LIN {X 0,Y 390.31,Z 233.363,A -85,B 0,C 180,E1 -11523.097,E2 -11523.097} C_VEL
LIN {X 0,Y 390.299,Z 233.363,A -85,B 0,C 180,E1 -11526.203,E2 -11526.203} C_VEL
LIN {X 0,Y 390.192,Z 233.354,A -85,B 0,C 180,E1 -11529.33,E2 -11529.33} C_VEL
LIN {X 0,Y 390.171,Z 233.375,A -85,B 0,C 180,E1 -11532.484,E2 -11532.484} C_VEL
LIN {X 0,Y 390.139,Z 233.38,A -85,B 0,C 180,E1 -11535.677,E2 -11535.677} C_VEL
LIN {X 0,Y 390.102,Z 233.369,A -85,B 0,C 180,E1 -11538.923,E2 -11538.923} C_VEL
LIN {X 0,Y 390.038,Z 233.396,A -85,B 0,C 180,E1 -11542.235,E2 -11542.235} C_VEL
LIN {X 0,Y 390.12,Z 233.376,A -85,B 0,C 180,E1 -11545.744,E2 -11545.744} C_VEL
LIN {X 0,Y 390.06,Z 233.395,A -85,B 0,C 180,E1 -11549.11,E2 -11549.11} C_VEL
LIN {X 0,Y 390.042,Z 233.39,A -85,B 0,C 180,E1 -11552.722,E2 -11552.722} C_VEL
LIN {X 0,Y 390.044,Z 233.392,A -85,B 0,C 180,E1 -11555.823,E2 -11555.823} C_VEL
LIN {X 0,Y 390.068,Z 233.387,A -85,B 0,C 180,E1 -11559.218,E2 -11559.218} C_VEL
LIN {X 0,Y 390.044,Z 233.403,A -85,B 0,C 180,E1 -11562.375,E2 -11562.375} C_VEL
LIN {X 0,Y 390.046,Z 233.395,A -85,B 0,C 180,E1 -11565.355,E2 -11565.355} C_VEL
LIN {X 0,Y 390.033,Z 233.39,A -85,B 0,C 180,E1 -11568.187,E2 -11568.187} C_VEL
LIN {X 0,Y 390.093,Z 233.385,A -85,B 0,C 180,E1 -11570.908,E2 -11570.908} C_VEL
LIN {X 0,Y 390.087,Z 233.384,A -85,B 0,C 180,E1 -11574.794,E2 -11574.794} C_VEL
LIN {X 0,Y 390.029,Z 233.399,A -85,B 0,C 180,E1 -11578.496,E2 -11578.496} C_VEL
LIN {X 0,Y 390.132,Z 233.546,A -85,B 0,C 180,E1 -11579.708,E2 -11579.708} C_VEL
LIN {X 0,Y 392.069,Z 243.393,A -85,B 0,C 180,E1 -11582.8,E2 -11582.8} C_VEL
LIN {X 0,Y 392.796,Z 249.65,A -85,B 0,C 180,E1 -11584.57,E2 -11584.57} C_VEL
LIN {X 0,Y 391.779,Z 261.902,A -85,B 0,C 180,E1 -11587.87,E2 -11587.87} C_VEL
LIN {X 0,Y 391.3,Z 267.747,A -85,B 0,C 180,E1 -11589.465,E2 -11589.465} C_VEL
LIN {X 0,Y 391.873,Z 270.886,A -85,B 0,C 180,E1 -11589.615,E2 -11589.615} C_VEL
LIN {X 0,Y 396.805,Z 298.116,A -85,B 0,C 180,E1 -11590.39,E2 -11590.39} C_VEL
LIN {X 0,Y 395.827,Z 372.67,A -85,B 0,C 180,E1 -11591.764,E2 -11591.764} C_VEL
LIN {X 0,Y 395.47,Z 383.442,A -85,B 0,C 180,E1 -11592.082,E2 -11592.082} C_VEL
LIN {X 0,Y 394.955,Z 392.542,A -85,B 0,C 180,E1 -11592.459,E2 -11592.459} C_VEL
LIN {X 0,Y 394.286,Z 402.904,A -85,B 0,C 180,E1 -11593.03,E2 -11593.03} C_VEL
LIN {X 0,Y 393.646,Z 412.039,A -85,B 0,C 180,E1 -11593.669,E2 -11593.669} C_VEL
LIN {X 0,Y 392.88,Z 421.035,A -85,B 0,C 180,E1 -11594.435,E2 -11594.435} C_VEL
LIN {X 0,Y 392.16,Z 429.764,A -85,B 0,C 180,E1 -11595.337,E2 -11595.337} C_VEL
LIN {X 0,Y 391.468,Z 437.493,A -85,B 0,C 180,E1 -11596.285,E2 -11596.285} C_VEL
LIN {X 0,Y 390.908,Z 444.382,A -85,B 0,C 180,E1 -11597.277,E2 -11597.277} C_VEL
LIN {X 0,Y 390.29,Z 450.582,A -85,B 0,C 180,E1 -11598.312,E2 -11598.312} C_VEL
LIN {X 0,Y 389.786,Z 457.122,A -85,B 0,C 180,E1 -11599.613,E2 -11599.613} C_VEL
LIN {X 0,Y 389.386,Z 461.622,A -85,B 0,C 180,E1 -11600.651,E2 -11600.651} C_VEL
LIN {X 0,Y 389.018,Z 467.114,A -85,B 0,C 180,E1 -11602.213,E2 -11602.213} C_VEL
LIN {X 0,Y 388.796,Z 471.439,A -85,B 0,C 180,E1 -11603.774,E2 -11603.774} C_VEL
LIN {X 0,Y 388.74,Z 473.806,A -85,B 0,C 180,E1 -11604.814,E2 -11604.814} C_VEL
LIN {X 0,Y 388.7,Z 475.604,A -85,B 0,C 180,E1 -11605.853,E2 -11605.853} C_VEL
LIN {X 0,Y 388.661,Z 478.048,A -85,B 0,C 180,E1 -11607.927,E2 -11607.927} C_VEL
LIN {X 0,Y 388.704,Z 478.637,A -85,B 0,C 180,E1 -11608.964,E2 -11608.964} C_VEL
LIN {X 0,Y 388.704,Z 478.637,A -85,B 0,C 180,E1 -11611.036,E2 -11611.036} C_VEL
LIN {X 0,Y 388.661,Z 478.048,A -85,B 0,C 180,E1 -11612.073,E2 -11612.073} C_VEL
LIN {X 0,Y 388.7,Z 475.604,A -85,B 0,C 180,E1 -11614.147,E2 -11614.147} C_VEL
LIN {X 0,Y 388.727,Z 472.551,A -85,B 0,C 180,E1 -11615.751,E2 -11615.751} C_VEL
LIN {X 0,Y 388.933,Z 468.668,A -85,B 0,C 180,E1 -11617.267,E2 -11617.267} C_VEL
LIN {X 0,Y 389.252,Z 463.539,A -85,B 0,C 180,E1 -11618.828,E2 -11618.828} C_VEL
LIN {X 0,Y 389.661,Z 458.277,A -85,B 0,C 180,E1 -11620.128,E2 -11620.128} C_VEL
LIN {X 0,Y 390.15,Z 451.958,A -85,B 0,C 180,E1 -11621.429,E2 -11621.429} C_VEL
LIN {X 0,Y 390.729,Z 446.008,A -85,B 0,C 180,E1 -11622.465,E2 -11622.465} C_VEL
LIN {X 0,Y 391.321,Z 439.079,A -85,B 0,C 180,E1 -11623.502,E2 -11623.502} C_VEL
LIN {X 0,Y 392.026,Z 430.898,A -85,B 0,C 180,E1 -11624.536,E2 -11624.536} C_VEL
LIN {X 0,Y 392.747,Z 422.386,A -85,B 0,C 180,E1 -11625.437,E2 -11625.437} C_VEL
LIN {X 0,Y 393.498,Z 413.67,A -85,B 0,C 180,E1 -11626.204,E2 -11626.204} C_VEL
LIN {X 0,Y 394.227,Z 403.912,A -85,B 0,C 180,E1 -11626.906,E2 -11626.906} C_VEL
LIN {X 0,Y 394.878,Z 393.83,A -85,B 0,C 180,E1 -11627.478,E2 -11627.478} C_VEL
LIN {X 0,Y 395.404,Z 384.315,A -85,B 0,C 180,E1 -11627.888,E2 -11627.888} C_VEL
LIN {X 0,Y 395.822,Z 374.003,A -85,B 0,C 180,E1 -11628.203,E2 -11628.203} C_VEL
LIN {X 0,Y 396.82,Z 301.34,A -85,B 0,C 180,E1 -11629.549,E2 -11629.549} C_VEL
LIN {X 0,Y 396.586,Z 296.789,A -85,B 0,C 180,E1 -11629.647,E2 -11629.647} C_VEL
LIN {X 0,Y 391.485,Z 269.134,A -85,B 0,C 180,E1 -11630.439,E2 -11630.439} C_VEL
LIN {X 0,Y 391.317,Z 267.542,A -85,B 0,C 180,E1 -11630.569,E2 -11630.569} C_VEL
LIN {X 0,Y 392.512,Z 253.975,A -85,B 0,C 180,E1 -11634.319,E2 -11634.319} C_VEL
LIN {X 0,Y 392.875,Z 249.939,A -85,B 0,C 180,E1 -11635.425,E2 -11635.425} C_VEL
LIN {X 0,Y 392.151,Z 243.762,A -85,B 0,C 180,E1 -11637.194,E2 -11637.194} C_VEL
LIN {X 0,Y 390.184,Z 233.887,A -85,B 0,C 180,E1 -11640.165,E2 -11640.165} C_VEL
LIN {X 0,Y 390.088,Z 233.399,A -85,B 0,C 180,E1 -11640.445,E2 -11640.445} C_VEL
LIN {X 0,Y 390.071,Z 233.398,A -85,B 0,C 180,E1 -11644.024,E2 -11644.024} C_VEL
LIN {X 0,Y 390.046,Z 233.4,A -85,B 0,C 180,E1 -11647.55,E2 -11647.55} C_VEL
LIN {X 0,Y 390.058,Z 233.377,A -85,B 0,C 180,E1 -11650.821,E2 -11650.821} C_VEL
LIN {X 0,Y 390.056,Z 233.398,A -85,B 0,C 180,E1 -11653.886,E2 -11653.886} C_VEL
LIN {X 0,Y 390.059,Z 233.394,A -85,B 0,C 180,E1 -11656.789,E2 -11656.789} C_VEL
LIN {X 0,Y 390.057,Z 233.39,A -85,B 0,C 180,E1 -11659.56,E2 -11659.56} C_VEL
LIN {X 0,Y 390.043,Z 233.397,A -85,B 0,C 180,E1 -11662.449,E2 -11662.449} C_VEL
LIN {X 0,Y 390.062,Z 233.383,A -85,B 0,C 180,E1 -11666.044,E2 -11666.044} C_VEL
LIN {X 0,Y 390.047,Z 233.397,A -85,B 0,C 180,E1 -11669.869,E2 -11669.869} C_VEL
LIN {X 0,Y 390.114,Z 233.372,A -85,B 0,C 180,E1 -11673.231,E2 -11673.231} C_VEL
LIN {X 0,Y 390.077,Z 233.392,A -85,B 0,C 180,E1 -11676.76,E2 -11676.76} C_VEL
LIN {X 0,Y 390.103,Z 233.375,A -85,B 0,C 180,E1 -11679.982,E2 -11679.982} C_VEL
LIN {X 0,Y 390.138,Z 233.375,A -85,B 0,C 180,E1 -11683.248,E2 -11683.248} C_VEL
LIN {X 0,Y 390.195,Z 233.378,A -85,B 0,C 180,E1 -11686.561,E2 -11686.561} C_VEL
LIN {X 0,Y 390.167,Z 233.358,A -85,B 0,C 180,E1 -11689.622,E2 -11689.622} C_VEL
LIN {X 0,Y 390.266,Z 233.36,A -85,B 0,C 180,E1 -11692.758,E2 -11692.758} C_VEL
LIN {X 0,Y 390.218,Z 233.379,A -85,B 0,C 180,E1 -11694.833,E2 -11694.833} C_VEL
LIN {X 0,Y 390.418,Z 233.343,A -85,B 0,C 180,E1 -11697.936,E2 -11697.936} C_VEL
LIN {X 0,Y 390.547,Z 233.31,A -85,B 0,C 180,E1 -11699.999,E2 -11699.999} C_VEL
LIN {X 0,Y 390.313,Z 233.362,A -85,B 0,C 180,E1 -11703.096,E2 -11703.096} C_VEL
LIN {X 0,Y 390.3,Z 233.362,A -85,B 0,C 180,E1 -11706.572,E2 -11706.572} C_VEL
LIN {X 0,Y 390.204,Z 233.353,A -85,B 0,C 180,E1 -11709.328,E2 -11709.328} C_VEL
LIN {X 0,Y 390.193,Z 233.377,A -85,B 0,C 180,E1 -11713.438,E2 -11713.438} C_VEL
LIN {X 0,Y 390.147,Z 233.374,A -85,B 0,C 180,E1 -11717.307,E2 -11717.307} C_VEL
LIN {X 0,Y 390.085,Z 233.379,A -85,B 0,C 180,E1 -11720.47,E2 -11720.47} C_VEL
LIN {X 0,Y 390.074,Z 233.393,A -85,B 0,C 180,E1 -11724.48,E2 -11724.48} C_VEL
LIN {X 0,Y 390.114,Z 233.371,A -85,B 0,C 180,E1 -11727.929,E2 -11727.929} C_VEL
LIN {X 0,Y 390.021,Z 233.401,A -85,B 0,C 180,E1 -11731.504,E2 -11731.504} C_VEL
LIN {X 0,Y 390.082,Z 233.382,A -85,B 0,C 180,E1 -11735.206,E2 -11735.206} C_VEL
LIN {X 0,Y 390.089,Z 233.39,A -85,B 0,C 180,E1 -11739.092,E2 -11739.092} C_VEL
LIN {X 0,Y 390.117,Z 233.39,A -85,B 0,C 180,E1 -11742.386,E2 -11742.386} C_VEL
LIN {X 0,Y 390.059,Z 233.389,A -85,B 0,C 180,E1 -11745.357,E2 -11745.357} C_VEL
LIN {X 0,Y 390.073,Z 233.371,A -85,B 0,C 180,E1 -11749.175,E2 -11749.175} C_VEL
LIN {X 0,Y 390.043,Z 233.398,A -85,B 0,C 180,E1 -11752.448,E2 -11752.448} C_VEL
LIN {X 0,Y 390.064,Z 233.377,A -85,B 0,C 180,E1 -11756.045,E2 -11756.045} C_VEL
LIN {X 0,Y 390.043,Z 233.386,A -85,B 0,C 180,E1 -11759.869,E2 -11759.869} C_VEL
LIN {X 0,Y 390.11,Z 233.394,A -85,B 0,C 180,E1 -11763.232,E2 -11763.232} C_VEL
LIN {X 0,Y 390.103,Z 233.393,A -85,B 0,C 180,E1 -11766.75,E2 -11766.75} C_VEL
LIN {X 0,Y 390.1,Z 233.395,A -85,B 0,C 180,E1 -11769.983,E2 -11769.983} C_VEL
LIN {X 0,Y 390.134,Z 233.391,A -85,B 0,C 180,E1 -11773.248,E2 -11773.248} C_VEL
LIN {X 0,Y 390.191,Z 233.383,A -85,B 0,C 180,E1 -11776.561,E2 -11776.561} C_VEL
LIN {X 0,Y 390.202,Z 233.382,A -85,B 0,C 180,E1 -11780.671,E2 -11780.671} C_VEL
LIN {X 0,Y 390.404,Z 233.767,A -85,B 0,C 180,E1 -11781.927,E2 -11781.927} C_VEL
LIN {X 0,Y 391.193,Z 235.98,A -85,B 0,C 180,E1 -11782.905,E2 -11782.905} C_VEL
LIN {X 0,Y 392.56,Z 237.719,A -85,B 0,C 180,E1 -11783.962,E2 -11783.962} C_VEL
LIN {X 0,Y 394.309,Z 239.002,A -85,B 0,C 180,E1 -11785.656,E2 -11785.656} C_VEL
LIN {X 0,Y 395.582,Z 239.492,A -85,B 0,C 180,E1 -11787.454,E2 -11787.454} C_VEL
LIN {X 0,Y 396.128,Z 239.931,A -85,B 0,C 180,E1 -11788.983,E2 -11788.983} C_VEL
LIN {X 0,Y 396.323,Z 239.849,A -85,B 0,C 180,E1 -11790,E2 -11790} C_VEL
LIN {X 0,Y 396.07,Z 239.804,A -85,B 0,C 180,E1 -11791.525,E2 -11791.525} C_VEL
LIN {X 0,Y 395.354,Z 239.371,A -85,B 0,C 180,E1 -11793.057,E2 -11793.057} C_VEL
LIN {X 0,Y 393.693,Z 238.657,A -85,B 0,C 180,E1 -11794.993,E2 -11794.993} C_VEL
LIN {X 0,Y 391.898,Z 237.018,A -85,B 0,C 180,E1 -11796.565,E2 -11796.565} C_VEL
LIN {X 0,Y 390.579,Z 234.501,A -85,B 0,C 180,E1 -11797.684,E2 -11797.684} C_VEL
LIN {X 0,Y 390.341,Z 233.593,A -85,B 0,C 180,E1 -11798.282,E2 -11798.282} C_VEL
LIN {X 0,Y 390.145,Z 233.389,A -85,B 0,C 180,E1 -11801.429,E2 -11801.429} C_VEL
LIN {X 0,Y 390.141,Z 233.39,A -85,B 0,C 180,E1 -11804.607,E2 -11804.607} C_VEL
LIN {X 0,Y 390.124,Z 233.392,A -85,B 0,C 180,E1 -11807.833,E2 -11807.833} C_VEL
LIN {X 0,Y 390.052,Z 233.401,A -85,B 0,C 180,E1 -11811.122,E2 -11811.122} C_VEL
LIN {X 0,Y 390.076,Z 233.398,A -85,B 0,C 180,E1 -11814.481,E2 -11814.481} C_VEL
LIN {X 0,Y 390.113,Z 233.387,A -85,B 0,C 180,E1 -11817.93,E2 -11817.93} C_VEL
LIN {X 0,Y 390.008,Z 233.394,A -85,B 0,C 180,E1 -11820.807,E2 -11820.807} C_VEL
LIN {X 0,Y 389.335,Z 233.489,A -85,B 0,C 180,E1 -11821.669,E2 -11821.669} C_VEL
LIN {X 0,Y 386.487,Z 233.835,A -85,B 0,C 180,E1 -11823.071,E2 -11823.071} C_VEL
LIN {X 0,Y 384.089,Z 234.122,A -85,B 0,C 180,E1 -11824.204,E2 -11824.204} C_VEL
LIN {X 0,Y 383.072,Z 234.245,A -85,B 0,C 180,E1 -11825.08,E2 -11825.08} C_VEL
LIN {X 0,Y 382.995,Z 234.255,A -85,B 0,C 180,E1 -11825.376,E2 -11825.376} C_VEL
LIN {X 0,Y 383.005,Z 234.275,A -85,B 0,C 180,E1 -11828.6,E2 -11828.6} C_VEL
LIN {X 0,Y 382.999,Z 234.243,A -85,B 0,C 180,E1 -11831.345,E2 -11831.345} C_VEL
LIN {X 0,Y 383.004,Z 234.261,A -85,B 0,C 180,E1 -11834.306,E2 -11834.306} C_VEL
LIN {X 0,Y 383.071,Z 234.266,A -85,B 0,C 180,E1 -11837.25,E2 -11837.25} C_VEL
LIN {X 0,Y 383.018,Z 234.27,A -85,B 0,C 180,E1 -11840.413,E2 -11840.413} C_VEL
LIN {X 0,Y 383.023,Z 234.266,A -85,B 0,C 180,E1 -11844.045,E2 -11844.045} C_VEL
LIN {X 0,Y 382.984,Z 234.275,A -85,B 0,C 180,E1 -11847.578,E2 -11847.578} C_VEL
LIN {X 0,Y 382.989,Z 234.273,A -85,B 0,C 180,E1 -11850.301,E2 -11850.301} C_VEL
LIN {X 0,Y 383.077,Z 234.256,A -85,B 0,C 180,E1 -11854.021,E2 -11854.021} C_VEL
LIN {X 0,Y 382.989,Z 234.279,A -85,B 0,C 180,E1 -11857.335,E2 -11857.335} C_VEL
LIN {X 0,Y 383.058,Z 234.245,A -85,B 0,C 180,E1 -11860.717,E2 -11860.717} C_VEL
LIN {X 0,Y 383.079,Z 234.265,A -85,B 0,C 180,E1 -11864.027,E2 -11864.027} C_VEL
LIN {X 0,Y 383.135,Z 234.255,A -85,B 0,C 180,E1 -11867.284,E2 -11867.284} C_VEL
LIN {X 0,Y 383.15,Z 234.231,A -85,B 0,C 180,E1 -11870.498,E2 -11870.498} C_VEL
LIN {X 0,Y 383.279,Z 234.242,A -85,B 0,C 180,E1 -11873.684,E2 -11873.684} C_VEL
LIN {X 0,Y 383.386,Z 234.213,A -85,B 0,C 180,E1 -11877.899,E2 -11877.899} C_VEL
LIN {X 0,Y 383.517,Z 234.184,A -85,B 0,C 180,E1 -11880.001,E2 -11880.001} C_VEL
LIN {X 0,Y 383.246,Z 234.243,A -85,B 0,C 180,E1 -11883.154,E2 -11883.154} C_VEL
LIN {X 0,Y 383.255,Z 234.24,A -85,B 0,C 180,E1 -11886.317,E2 -11886.317} C_VEL
LIN {X 0,Y 383.143,Z 234.231,A -85,B 0,C 180,E1 -11889.503,E2 -11889.503} C_VEL
LIN {X 0,Y 383.136,Z 234.253,A -85,B 0,C 180,E1 -11892.717,E2 -11892.717} C_VEL
LIN {X 0,Y 383.081,Z 234.259,A -85,B 0,C 180,E1 -11895.974,E2 -11895.974} C_VEL
LIN {X 0,Y 383.058,Z 234.248,A -85,B 0,C 180,E1 -11899.284,E2 -11899.284} C_VEL
LIN {X 0,Y 382.996,Z 234.277,A -85,B 0,C 180,E1 -11902.666,E2 -11902.666} C_VEL
LIN {X 0,Y 383.08,Z 234.251,A -85,B 0,C 180,E1 -11906.124,E2 -11906.124} C_VEL
LIN {X 0,Y 382.993,Z 234.274,A -85,B 0,C 180,E1 -11909.7,E2 -11909.7} C_VEL
LIN {X 0,Y 382.999,Z 234.262,A -85,B 0,C 180,E1 -11913.402,E2 -11913.402} C_VEL
LIN {X 0,Y 383.024,Z 234.269,A -85,B 0,C 180,E1 -11916.163,E2 -11916.163} C_VEL
LIN {X 0,Y 383.009,Z 234.266,A -85,B 0,C 180,E1 -11919.959,E2 -11919.959} C_VEL
LIN {X 0,Y 383.007,Z 234.275,A -85,B 0,C 180,E1 -11922.779,E2 -11922.779} C_VEL
LIN {X 0,Y 382.999,Z 234.275,A -85,B 0,C 180,E1 -11925.79,E2 -11925.79} C_VEL
LIN {X 0,Y 382.99,Z 234.26,A -85,B 0,C 180,E1 -11928.796,E2 -11928.796} C_VEL
LIN {X 0,Y 383.002,Z 234.279,A -85,B 0,C 180,E1 -11932.097,E2 -11932.097} C_VEL
LIN {X 0,Y 383.02,Z 234.269,A -85,B 0,C 180,E1 -11935.332,E2 -11935.332} C_VEL
LIN {X 0,Y 383.049,Z 234.292,A -85,B 0,C 180,E1 -11939.309,E2 -11939.309} C_VEL
LIN {X 0,Y 384.788,Z 243.209,A -85,B 0,C 180,E1 -11942.242,E2 -11942.242} C_VEL
LIN {X 0,Y 385.782,Z 249.475,A -85,B 0,C 180,E1 -11944.073,E2 -11944.073} C_VEL
LIN {X 0,Y 385.378,Z 256.646,A -85,B 0,C 180,E1 -11946.036,E2 -11946.036} C_VEL
LIN {X 0,Y 384.406,Z 267.552,A -85,B 0,C 180,E1 -11949.078,E2 -11949.078} C_VEL
LIN {X 0,Y 384.82,Z 270.202,A -85,B 0,C 180,E1 -11949.215,E2 -11949.215} C_VEL
LIN {X 0,Y 390.06,Z 298.316,A -85,B 0,C 180,E1 -11950.044,E2 -11950.044} C_VEL
LIN {X 0,Y 389.103,Z 372.478,A -85,B 0,C 180,E1 -11951.437,E2 -11951.437} C_VEL
LIN {X 0,Y 388.708,Z 383.249,A -85,B 0,C 180,E1 -11951.759,E2 -11951.759} C_VEL
LIN {X 0,Y 388.182,Z 392.349,A -85,B 0,C 180,E1 -11952.143,E2 -11952.143} C_VEL
LIN {X 0,Y 387.492,Z 402.711,A -85,B 0,C 180,E1 -11952.723,E2 -11952.723} C_VEL
LIN {X 0,Y 386.841,Z 411.846,A -85,B 0,C 180,E1 -11953.373,E2 -11953.373} C_VEL
LIN {X 0,Y 386.018,Z 420.841,A -85,B 0,C 180,E1 -11954.151,E2 -11954.151} C_VEL
LIN {X 0,Y 385.273,Z 429.571,A -85,B 0,C 180,E1 -11955.069,E2 -11955.069} C_VEL
LIN {X 0,Y 384.536,Z 437.481,A -85,B 0,C 180,E1 -11956.058,E2 -11956.058} C_VEL
LIN {X 0,Y 383.792,Z 445.815,A -85,B 0,C 180,E1 -11957.306,E2 -11957.306} C_VEL
LIN {X 0,Y 383.166,Z 451.764,A -85,B 0,C 180,E1 -11958.36,E2 -11958.36} C_VEL
LIN {X 0,Y 382.657,Z 458.083,A -85,B 0,C 180,E1 -11959.684,E2 -11959.684} C_VEL
LIN {X 0,Y 382.209,Z 463.345,A -85,B 0,C 180,E1 -11961.008,E2 -11961.008} C_VEL
LIN {X 0,Y 381.861,Z 468.474,A -85,B 0,C 180,E1 -11962.598,E2 -11962.598} C_VEL
LIN {X 0,Y 381.688,Z 471.762,A -85,B 0,C 180,E1 -11963.883,E2 -11963.883} C_VEL
LIN {X 0,Y 381.641,Z 473.612,A -85,B 0,C 180,E1 -11964.717,E2 -11964.717} C_VEL
LIN {X 0,Y 381.625,Z 475.411,A -85,B 0,C 180,E1 -11965.776,E2 -11965.776} C_VEL
LIN {X 0,Y 381.56,Z 477.855,A -85,B 0,C 180,E1 -11967.889,E2 -11967.889} C_VEL
LIN {X 0,Y 381.603,Z 478.444,A -85,B 0,C 180,E1 -11968.945,E2 -11968.945} C_VEL
LIN {X 0,Y 381.603,Z 478.444,A -85,B 0,C 180,E1 -11971.055,E2 -11971.055} C_VEL
LIN {X 0,Y 381.56,Z 477.855,A -85,B 0,C 180,E1 -11972.111,E2 -11972.111} C_VEL
LIN {X 0,Y 381.625,Z 475.411,A -85,B 0,C 180,E1 -11974.224,E2 -11974.224} C_VEL
LIN {X 0,Y 381.641,Z 473.612,A -85,B 0,C 180,E1 -11975.283,E2 -11975.283} C_VEL
LIN {X 0,Y 381.781,Z 470.005,A -85,B 0,C 180,E1 -11976.872,E2 -11976.872} C_VEL
LIN {X 0,Y 382.058,Z 465.26,A -85,B 0,C 180,E1 -11978.462,E2 -11978.462} C_VEL
LIN {X 0,Y 382.532,Z 459.238,A -85,B 0,C 180,E1 -11980.052,E2 -11980.052} C_VEL
LIN {X 0,Y 383.05,Z 453.141,A -85,B 0,C 180,E1 -11981.375,E2 -11981.375} C_VEL
LIN {X 0,Y 383.611,Z 447.441,A -85,B 0,C 180,E1 -11982.431,E2 -11982.431} C_VEL
LIN {X 0,Y 384.39,Z 438.886,A -85,B 0,C 180,E1 -11983.75,E2 -11983.75} C_VEL
LIN {X 0,Y 385.145,Z 430.705,A -85,B 0,C 180,E1 -11984.801,E2 -11984.801} C_VEL
LIN {X 0,Y 385.907,Z 422.193,A -85,B 0,C 180,E1 -11985.718,E2 -11985.718} C_VEL
LIN {X 0,Y 386.667,Z 413.477,A -85,B 0,C 180,E1 -11986.499,E2 -11986.499} C_VEL
LIN {X 0,Y 387.429,Z 403.719,A -85,B 0,C 180,E1 -11987.212,E2 -11987.212} C_VEL
LIN {X 0,Y 388.121,Z 393.637,A -85,B 0,C 180,E1 -11987.792,E2 -11987.792} C_VEL
LIN {X 0,Y 388.668,Z 384.123,A -85,B 0,C 180,E1 -11988.209,E2 -11988.209} C_VEL
LIN {X 0,Y 389.092,Z 373.81,A -85,B 0,C 180,E1 -11988.529,E2 -11988.529} C_VEL
LIN {X 0,Y 390.142,Z 301.313,A -85,B 0,C 180,E1 -11989.895,E2 -11989.895} C_VEL
LIN {X 0,Y 389.76,Z 296.708,A -85,B 0,C 180,E1 -11990.003,E2 -11990.003} C_VEL
LIN {X 0,Y 384.568,Z 268.933,A -85,B 0,C 180,E1 -11990.824,E2 -11990.824} C_VEL
LIN {X 0,Y 384.385,Z 267.342,A -85,B 0,C 180,E1 -11990.958,E2 -11990.958} C_VEL
LIN {X 0,Y 385.663,Z 253.791,A -85,B 0,C 180,E1 -11994.78,E2 -11994.78} C_VEL
LIN {X 0,Y 385.873,Z 249.767,A -85,B 0,C 180,E1 -11995.92,E2 -11995.92} C_VEL
LIN {X 0,Y 384.556,Z 241.517,A -85,B 0,C 180,E1 -11998.37,E2 -11998.37} C_VEL
LIN {X 0,Y 383.049,Z 234.295,A -85,B 0,C 180,E1 -12000.692,E2 -12000.692} C_VEL
LIN {X 0,Y 383.02,Z 234.27,A -85,B 0,C 180,E1 -12004.668,E2 -12004.668} C_VEL
LIN {X 0,Y 383.002,Z 234.279,A -85,B 0,C 180,E1 -12007.903,E2 -12007.903} C_VEL
LIN {X 0,Y 382.985,Z 234.261,A -85,B 0,C 180,E1 -12011.347,E2 -12011.347} C_VEL
LIN {X 0,Y 382.997,Z 234.274,A -85,B 0,C 180,E1 -12014.303,E2 -12014.303} C_VEL
LIN {X 0,Y 383.012,Z 234.274,A -85,B 0,C 180,E1 -12017.24,E2 -12017.24} C_VEL
LIN {X 0,Y 383.015,Z 234.266,A -85,B 0,C 180,E1 -12020.413,E2 -12020.413} C_VEL
LIN {X 0,Y 383.016,Z 234.269,A -85,B 0,C 180,E1 -12024.043,E2 -12024.043} C_VEL
LIN {X 0,Y 382.986,Z 234.273,A -85,B 0,C 180,E1 -12027.578,E2 -12027.578} C_VEL
LIN {X 0,Y 382.993,Z 234.274,A -85,B 0,C 180,E1 -12030.3,E2 -12030.3} C_VEL
LIN {X 0,Y 383.081,Z 234.253,A -85,B 0,C 180,E1 -12034.02,E2 -12034.02} C_VEL
LIN {X 0,Y 382.996,Z 234.277,A -85,B 0,C 180,E1 -12037.334,E2 -12037.334} C_VEL
LIN {X 0,Y 383.058,Z 234.248,A -85,B 0,C 180,E1 -12040.716,E2 -12040.716} C_VEL
LIN {X 0,Y 383.081,Z 234.259,A -85,B 0,C 180,E1 -12044.026,E2 -12044.026} C_VEL
LIN {X 0,Y 383.136,Z 234.253,A -85,B 0,C 180,E1 -12047.283,E2 -12047.283} C_VEL
LIN {X 0,Y 383.143,Z 234.231,A -85,B 0,C 180,E1 -12050.497,E2 -12050.497} C_VEL
LIN {X 0,Y 383.255,Z 234.24,A -85,B 0,C 180,E1 -12053.683,E2 -12053.683} C_VEL
LIN {X 0,Y 383.385,Z 234.218,A -85,B 0,C 180,E1 -12057.898,E2 -12057.898} C_VEL
LIN {X 0,Y 383.517,Z 234.184,A -85,B 0,C 180,E1 -12059.999,E2 -12059.999} C_VEL
LIN {X 0,Y 383.249,Z 234.243,A -85,B 0,C 180,E1 -12063.153,E2 -12063.153} C_VEL
LIN {X 0,Y 383.261,Z 234.24,A -85,B 0,C 180,E1 -12066.563,E2 -12066.563} C_VEL
LIN {X 0,Y 383.15,Z 234.231,A -85,B 0,C 180,E1 -12069.502,E2 -12069.502} C_VEL
LIN {X 0,Y 383.124,Z 234.257,A -85,B 0,C 180,E1 -12073.536,E2 -12073.536} C_VEL
LIN {X 0,Y 383.093,Z 234.253,A -85,B 0,C 180,E1 -12077.454,E2 -12077.454} C_VEL
LIN {X 0,Y 383.026,Z 234.26,A -85,B 0,C 180,E1 -12080.646,E2 -12080.646} C_VEL
LIN {X 0,Y 383.02,Z 234.274,A -85,B 0,C 180,E1 -12083.807,E2 -12083.807} C_VEL
LIN {X 0,Y 383.077,Z 234.254,A -85,B 0,C 180,E1 -12086.123,E2 -12086.123} C_VEL
LIN {X 0,Y 382.989,Z 234.273,A -85,B 0,C 180,E1 -12089.699,E2 -12089.699} C_VEL
LIN {X 0,Y 383,Z 234.27,A -85,B 0,C 180,E1 -12093.4,E2 -12093.4} C_VEL
LIN {X 0,Y 383.03,Z 234.268,A -85,B 0,C 180,E1 -12096.164,E2 -12096.164} C_VEL
LIN {X 0,Y 383.014,Z 234.266,A -85,B 0,C 180,E1 -12099.957,E2 -12099.957} C_VEL
LIN {X 0,Y 383.062,Z 234.267,A -85,B 0,C 180,E1 -12102.788,E2 -12102.788} C_VEL
LIN {X 0,Y 383.004,Z 234.259,A -85,B 0,C 180,E1 -12105.79,E2 -12105.79} C_VEL
LIN {X 0,Y 383.004,Z 234.244,A -85,B 0,C 180,E1 -12108.792,E2 -12108.792} C_VEL
LIN {X 0,Y 382.999,Z 234.278,A -85,B 0,C 180,E1 -12112.095,E2 -12112.095} C_VEL
LIN {X 0,Y 383.014,Z 234.251,A -85,B 0,C 180,E1 -12115.332,E2 -12115.332} C_VEL
LIN {X 0,Y 382.979,Z 234.278,A -85,B 0,C 180,E1 -12119.081,E2 -12119.081} C_VEL
LIN {X 0,Y 383.053,Z 234.27,A -85,B 0,C 180,E1 -12122.698,E2 -12122.698} C_VEL
LIN {X 0,Y 383.03,Z 234.274,A -85,B 0,C 180,E1 -12126.193,E2 -12126.193} C_VEL
LIN {X 0,Y 383.051,Z 234.273,A -85,B 0,C 180,E1 -12129.598,E2 -12129.598} C_VEL
LIN {X 0,Y 383.101,Z 234.267,A -85,B 0,C 180,E1 -12132.931,E2 -12132.931} C_VEL
LIN {X 0,Y 383.121,Z 234.263,A -85,B 0,C 180,E1 -12136.464,E2 -12136.464} C_VEL
LIN {X 0,Y 383.154,Z 234.531,A -85,B 0,C 180,E1 -12138.527,E2 -12138.527} C_VEL
LIN {X 0,Y 383.436,Z 235.716,A -85,B 0,C 180,E1 -12138.971,E2 -12138.971} C_VEL
LIN {X 0,Y 384.578,Z 237.759,A -85,B 0,C 180,E1 -12139.603,E2 -12139.603} C_VEL
LIN {X 0,Y 386.856,Z 239.64,A -85,B 0,C 180,E1 -12140.722,E2 -12140.722} C_VEL
LIN {X 0,Y 388.921,Z 240.829,A -85,B 0,C 180,E1 -12141.896,E2 -12141.896} C_VEL
LIN {X 0,Y 390.34,Z 243.395,A -85,B 0,C 180,E1 -12142.955,E2 -12142.955} C_VEL
LIN {X 0,Y 391.933,Z 245.07,A -85,B 0,C 180,E1 -12144.211,E2 -12144.211} C_VEL
LIN {X 0,Y 393.437,Z 246.033,A -85,B 0,C 180,E1 -12145.646,E2 -12145.646} C_VEL
LIN {X 0,Y 394.719,Z 246.512,A -85,B 0,C 180,E1 -12147.449,E2 -12147.449} C_VEL
LIN {X 0,Y 395.266,Z 246.977,A -85,B 0,C 180,E1 -12148.981,E2 -12148.981} C_VEL
LIN {X 0,Y 395.458,Z 246.896,A -85,B 0,C 180,E1 -12150,E2 -12150} C_VEL
LIN {X 0,Y 395.202,Z 246.853,A -85,B 0,C 180,E1 -12151.529,E2 -12151.529} C_VEL
LIN {X 0,Y 394.244,Z 246.355,A -85,B 0,C 180,E1 -12153.368,E2 -12153.368} C_VEL
LIN {X 0,Y 392.65,Z 245.62,A -85,B 0,C 180,E1 -12155.135,E2 -12155.135} C_VEL
LIN {X 0,Y 390.787,Z 243.978,A -85,B 0,C 180,E1 -12156.713,E2 -12156.713} C_VEL
LIN {X 0,Y 389.246,Z 241.409,A -85,B 0,C 180,E1 -12157.901,E2 -12157.901} C_VEL
LIN {X 0,Y 388.306,Z 240.316,A -85,B 0,C 180,E1 -12158.456,E2 -12158.456} C_VEL
LIN {X 0,Y 385.837,Z 239.007,A -85,B 0,C 180,E1 -12159.766,E2 -12159.766} C_VEL
LIN {X 0,Y 383.934,Z 236.786,A -85,B 0,C 180,E1 -12160.748,E2 -12160.748} C_VEL
LIN {X 0,Y 383.222,Z 234.963,A -85,B 0,C 180,E1 -12161.236,E2 -12161.236} C_VEL
LIN {X 0,Y 383.115,Z 234.297,A -85,B 0,C 180,E1 -12161.91,E2 -12161.91} C_VEL
LIN {X 0,Y 383.107,Z 234.266,A -85,B 0,C 180,E1 -12164.882,E2 -12164.882} C_VEL
LIN {X 0,Y 383.086,Z 234.268,A -85,B 0,C 180,E1 -12168.172,E2 -12168.172} C_VEL
LIN {X 0,Y 382.989,Z 234.279,A -85,B 0,C 180,E1 -12171.531,E2 -12171.531} C_VEL
LIN {X 0,Y 383.049,Z 234.272,A -85,B 0,C 180,E1 -12174.96,E2 -12174.96} C_VEL
LIN {X 0,Y 383.013,Z 234.26,A -85,B 0,C 180,E1 -12178.495,E2 -12178.495} C_VEL
LIN {X 0,Y 383.006,Z 234.278,A -85,B 0,C 180,E1 -12182.15,E2 -12182.15} C_VEL
LIN {X 0,Y 382.995,Z 234.255,A -85,B 0,C 180,E1 -12185.376,E2 -12185.376} C_VEL
LIN {X 0,Y 382.355,Z 234.346,A -85,B 0,C 180,E1 -12186.254,E2 -12186.254} C_VEL
LIN {X 0,Y 379.55,Z 234.706,A -85,B 0,C 180,E1 -12187.682,E2 -12187.682} C_VEL
LIN {X 0,Y 377.146,Z 235.004,A -85,B 0,C 180,E1 -12188.836,E2 -12188.836} C_VEL
LIN {X 0,Y 376.089,Z 235.127,A -85,B 0,C 180,E1 -12189.728,E2 -12189.728} C_VEL
LIN {X 0,Y 375.989,Z 235.133,A -85,B 0,C 180,E1 -12190.031,E2 -12190.031} C_VEL
LIN {X 0,Y 375.933,Z 235.134,A -85,B 0,C 180,E1 -12193.765,E2 -12193.765} C_VEL
LIN {X 0,Y 375.986,Z 235.149,A -85,B 0,C 180,E1 -12196.802,E2 -12196.802} C_VEL
LIN {X 0,Y 375.995,Z 235.14,A -85,B 0,C 180,E1 -12200.028,E2 -12200.028} C_VEL
LIN {X 0,Y 375.962,Z 235.154,A -85,B 0,C 180,E1 -12203.496,E2 -12203.496} C_VEL
LIN {X 0,Y 375.957,Z 235.14,A -85,B 0,C 180,E1 -12205.889,E2 -12205.889} C_VEL
LIN {X 0,Y 375.961,Z 235.155,A -85,B 0,C 180,E1 -12209.688,E2 -12209.688} C_VEL
LIN {X 0,Y 376.017,Z 235.126,A -85,B 0,C 180,E1 -12213.348,E2 -12213.348} C_VEL
LIN {X 0,Y 375.976,Z 235.15,A -85,B 0,C 180,E1 -12216.888,E2 -12216.888} C_VEL
LIN {X 0,Y 375.995,Z 235.125,A -85,B 0,C 180,E1 -12220.34,E2 -12220.34} C_VEL
LIN {X 0,Y 376.028,Z 235.142,A -85,B 0,C 180,E1 -12223.719,E2 -12223.719} C_VEL
LIN {X 0,Y 376.102,Z 235.134,A -85,B 0,C 180,E1 -12227.043,E2 -12227.043} C_VEL
LIN {X 0,Y 376.118,Z 235.106,A -85,B 0,C 180,E1 -12230.319,E2 -12230.319} C_VEL
LIN {X 0,Y 376.237,Z 235.119,A -85,B 0,C 180,E1 -12233.565,E2 -12233.565} C_VEL
LIN {X 0,Y 376.352,Z 235.089,A -85,B 0,C 180,E1 -12237.86,E2 -12237.86} C_VEL
LIN {X 0,Y 376.486,Z 235.059,A -85,B 0,C 180,E1 -12240.001,E2 -12240.001} C_VEL
LIN {X 0,Y 376.184,Z 235.123,A -85,B 0,C 180,E1 -12243.214,E2 -12243.214} C_VEL
LIN {X 0,Y 376.213,Z 235.118,A -85,B 0,C 180,E1 -12246.436,E2 -12246.436} C_VEL
LIN {X 0,Y 376.113,Z 235.106,A -85,B 0,C 180,E1 -12249.682,E2 -12249.682} C_VEL
LIN {X 0,Y 376.089,Z 235.133,A -85,B 0,C 180,E1 -12253.658,E2 -12253.658} C_VEL
LIN {X 0,Y 376.032,Z 235.124,A -85,B 0,C 180,E1 -12257.4,E2 -12257.4} C_VEL
LIN {X 0,Y 375.979,Z 235.141,A -85,B 0,C 180,E1 -12260.833,E2 -12260.833} C_VEL
LIN {X 0,Y 375.99,Z 235.148,A -85,B 0,C 180,E1 -12264.282,E2 -12264.282} C_VEL
LIN {X 0,Y 376.02,Z 235.126,A -85,B 0,C 180,E1 -12266.653,E2 -12266.653} C_VEL
LIN {X 0,Y 375.965,Z 235.153,A -85,B 0,C 180,E1 -12270.313,E2 -12270.313} C_VEL
LIN {X 0,Y 375.958,Z 235.138,A -85,B 0,C 180,E1 -12274.112,E2 -12274.112} C_VEL
LIN {X 0,Y 375.951,Z 235.156,A -85,B 0,C 180,E1 -12276.742,E2 -12276.742} C_VEL
LIN {X 0,Y 375.989,Z 235.14,A -85,B 0,C 180,E1 -12279.971,E2 -12279.971} C_VEL
LIN {X 0,Y 375.931,Z 235.155,A -85,B 0,C 180,E1 -12283.766,E2 -12283.766} C_VEL
LIN {X 0,Y 375.936,Z 235.156,A -85,B 0,C 180,E1 -12286.811,E2 -12286.811} C_VEL
LIN {X 0,Y 375.965,Z 235.137,A -85,B 0,C 180,E1 -12290.538,E2 -12290.538} C_VEL
LIN {X 0,Y 375.966,Z 235.145,A -85,B 0,C 180,E1 -12293.496,E2 -12293.496} C_VEL
LIN {X 0,Y 375.963,Z 235.154,A -85,B 0,C 180,E1 -12295.889,E2 -12295.889} C_VEL
LIN {X 0,Y 376.016,Z 235.337,A -85,B 0,C 180,E1 -12299.1,E2 -12299.1} C_VEL
LIN {X 0,Y 377.966,Z 245.117,A -85,B 0,C 180,E1 -12302.299,E2 -12302.299} C_VEL
LIN {X 0,Y 378.867,Z 251.381,A -85,B 0,C 180,E1 -12304.156,E2 -12304.156} C_VEL
LIN {X 0,Y 378.192,Z 259.568,A -85,B 0,C 180,E1 -12306.451,E2 -12306.451} C_VEL
LIN {X 0,Y 377.468,Z 267.424,A -85,B 0,C 180,E1 -12308.686,E2 -12308.686} C_VEL
LIN {X 0,Y 378.455,Z 272.569,A -85,B 0,C 180,E1 -12308.9,E2 -12308.9} C_VEL
LIN {X 0,Y 383.441,Z 299.914,A -85,B 0,C 180,E1 -12309.719,E2 -12309.719} C_VEL
LIN {X 0,Y 382.381,Z 372.285,A -85,B 0,C 180,E1 -12311.099,E2 -12311.099} C_VEL
LIN {X 0,Y 381.981,Z 383.056,A -85,B 0,C 180,E1 -12311.426,E2 -12311.426} C_VEL
LIN {X 0,Y 381.439,Z 392.156,A -85,B 0,C 180,E1 -12311.816,E2 -12311.816} C_VEL
LIN {X 0,Y 380.772,Z 401.511,A -85,B 0,C 180,E1 -12312.339,E2 -12312.339} C_VEL
LIN {X 0,Y 380.035,Z 411.653,A -85,B 0,C 180,E1 -12313.066,E2 -12313.066} C_VEL
LIN {X 0,Y 379.197,Z 420.649,A -85,B 0,C 180,E1 -12313.859,E2 -12313.859} C_VEL
LIN {X 0,Y 378.392,Z 429.378,A -85,B 0,C 180,E1 -12314.791,E2 -12314.791} C_VEL
LIN {X 0,Y 377.615,Z 437.473,A -85,B 0,C 180,E1 -12315.824,E2 -12315.824} C_VEL
LIN {X 0,Y 376.841,Z 445.621,A -85,B 0,C 180,E1 -12317.068,E2 -12317.068} C_VEL
LIN {X 0,Y 376.195,Z 451.571,A -85,B 0,C 180,E1 -12318.141,E2 -12318.141} C_VEL
LIN {X 0,Y 375.645,Z 457.89,A -85,B 0,C 180,E1 -12319.49,E2 -12319.49} C_VEL
LIN {X 0,Y 375.165,Z 463.151,A -85,B 0,C 180,E1 -12320.838,E2 -12320.838} C_VEL
LIN {X 0,Y 374.794,Z 468.281,A -85,B 0,C 180,E1 -12322.458,E2 -12322.458} C_VEL
LIN {X 0,Y 374.583,Z 471.95,A -85,B 0,C 180,E1 -12323.936,E2 -12323.936} C_VEL
LIN {X 0,Y 374.53,Z 475.218,A -85,B 0,C 180,E1 -12325.695,E2 -12325.695} C_VEL
LIN {X 0,Y 374.459,Z 477.662,A -85,B 0,C 180,E1 -12327.849,E2 -12327.849} C_VEL
LIN {X 0,Y 374.503,Z 478.252,A -85,B 0,C 180,E1 -12328.925,E2 -12328.925} C_VEL
LIN {X 0,Y 374.503,Z 478.252,A -85,B 0,C 180,E1 -12331.075,E2 -12331.075} C_VEL
LIN {X 0,Y 374.459,Z 477.662,A -85,B 0,C 180,E1 -12332.151,E2 -12332.151} C_VEL
LIN {X 0,Y 374.53,Z 475.218,A -85,B 0,C 180,E1 -12334.305,E2 -12334.305} C_VEL
LIN {X 0,Y 374.583,Z 471.951,A -85,B 0,C 180,E1 -12336.064,E2 -12336.064} C_VEL
LIN {X 0,Y 374.794,Z 468.281,A -85,B 0,C 180,E1 -12337.542,E2 -12337.542} C_VEL
LIN {X 0,Y 375.165,Z 463.151,A -85,B 0,C 180,E1 -12339.162,E2 -12339.162} C_VEL
LIN {X 0,Y 375.645,Z 457.89,A -85,B 0,C 180,E1 -12340.51,E2 -12340.51} C_VEL
LIN {X 0,Y 376.193,Z 451.571,A -85,B 0,C 180,E1 -12341.859,E2 -12341.859} C_VEL
LIN {X 0,Y 376.832,Z 445.621,A -85,B 0,C 180,E1 -12342.932,E2 -12342.932} C_VEL
LIN {X 0,Y 377.609,Z 437.479,A -85,B 0,C 180,E1 -12344.176,E2 -12344.176} C_VEL
LIN {X 0,Y 378.498,Z 428.243,A -85,B 0,C 180,E1 -12345.343,E2 -12345.343} C_VEL
LIN {X 0,Y 379.497,Z 417.947,A -85,B 0,C 180,E1 -12346.405,E2 -12346.405} C_VEL
LIN {X 0,Y 380.504,Z 405.54,A -85,B 0,C 180,E1 -12347.397,E2 -12347.397} C_VEL
LIN {X 0,Y 381.286,Z 394.732,A -85,B 0,C 180,E1 -12348.053,E2 -12348.053} C_VEL
LIN {X 0,Y 381.902,Z 384.805,A -85,B 0,C 180,E1 -12348.508,E2 -12348.508} C_VEL
LIN {X 0,Y 382.323,Z 374.949,A -85,B 0,C 180,E1 -12348.835,E2 -12348.835} C_VEL
LIN {X 0,Y 382.777,Z 349.31,A -85,B 0,C 180,E1 -12349.353,E2 -12349.353} C_VEL
LIN {X 0,Y 383.333,Z 299.183,A -85,B 0,C 180,E1 -12350.301,E2 -12350.301} C_VEL
LIN {X 0,Y 378.322,Z 271.829,A -85,B 0,C 180,E1 -12351.123,E2 -12351.123} C_VEL
LIN {X 0,Y 377.499,Z 267.585,A -85,B 0,C 180,E1 -12351.292,E2 -12351.292} C_VEL
LIN {X 0,Y 377.615,Z 265.391,A -85,B 0,C 180,E1 -12351.853,E2 -12351.853} C_VEL
LIN {X 0,Y 378.927,Z 252.607,A -85,B 0,C 180,E1 -12355.545,E2 -12355.545} C_VEL
LIN {X 0,Y 378.516,Z 247.831,A -85,B 0,C 180,E1 -12356.971,E2 -12356.971} C_VEL
LIN {X 0,Y 376.421,Z 237.193,A -85,B 0,C 180,E1 -12360.272,E2 -12360.272} C_VEL
LIN {X 0,Y 375.988,Z 235.17,A -85,B 0,C 180,E1 -12361.025,E2 -12361.025} C_VEL
LIN {X 0,Y 375.982,Z 235.146,A -85,B 0,C 180,E1 -12364.667,E2 -12364.667} C_VEL
LIN {X 0,Y 375.976,Z 235.15,A -85,B 0,C 180,E1 -12368.27,E2 -12368.27} C_VEL
LIN {X 0,Y 375.936,Z 235.141,A -85,B 0,C 180,E1 -12371.6,E2 -12371.6} C_VEL
LIN {X 0,Y 375.928,Z 235.152,A -85,B 0,C 180,E1 -12375.268,E2 -12375.268} C_VEL
LIN {X 0,Y 375.935,Z 235.153,A -85,B 0,C 180,E1 -12378.399,E2 -12378.399} C_VEL
LIN {X 0,Y 375.973,Z 235.152,A -85,B 0,C 180,E1 -12381.729,E2 -12381.729} C_VEL
LIN {X 0,Y 375.975,Z 235.138,A -85,B 0,C 180,E1 -12385.333,E2 -12385.333} C_VEL
LIN {X 0,Y 375.958,Z 235.151,A -85,B 0,C 180,E1 -12388.437,E2 -12388.437} C_VEL
LIN {X 0,Y 375.984,Z 235.134,A -85,B 0,C 180,E1 -12392.14,E2 -12392.14} C_VEL
LIN {X 0,Y 376.006,Z 235.134,A -85,B 0,C 180,E1 -12394.538,E2 -12394.538} C_VEL
LIN {X 0,Y 375.958,Z 235.148,A -85,B 0,C 180,E1 -12398.045,E2 -12398.045} C_VEL
LIN {X 0,Y 376.002,Z 235.123,A -85,B 0,C 180,E1 -12401.472,E2 -12401.472} C_VEL
LIN {X 0,Y 376.058,Z 235.137,A -85,B 0,C 180,E1 -12404.832,E2 -12404.832} C_VEL
LIN {X 0,Y 376.049,Z 235.131,A -85,B 0,C 180,E1 -12408.136,E2 -12408.136} C_VEL
LIN {X 0,Y 376.193,Z 235.108,A -85,B 0,C 180,E1 -12411.946,E2 -12411.946} C_VEL
LIN {X 0,Y 376.16,Z 235.127,A -85,B 0,C 180,E1 -12414.639,E2 -12414.639} C_VEL
LIN {X 0,Y 376.351,Z 235.094,A -85,B 0,C 180,E1 -12417.859,E2 -12417.859} C_VEL
LIN {X 0,Y 376.486,Z 235.059,A -85,B 0,C 180,E1 -12419.999,E2 -12419.999} C_VEL
LIN {X 0,Y 376.187,Z 235.122,A -85,B 0,C 180,E1 -12423.212,E2 -12423.212} C_VEL
LIN {X 0,Y 376.227,Z 235.118,A -85,B 0,C 180,E1 -12426.55,E2 -12426.55} C_VEL
LIN {X 0,Y 376.118,Z 235.106,A -85,B 0,C 180,E1 -12429.681,E2 -12429.681} C_VEL
LIN {X 0,Y 376.088,Z 235.134,A -85,B 0,C 180,E1 -12433.657,E2 -12433.657} C_VEL
LIN {X 0,Y 376.041,Z 235.131,A -85,B 0,C 180,E1 -12437.606,E2 -12437.606} C_VEL
LIN {X 0,Y 375.976,Z 235.141,A -85,B 0,C 180,E1 -12440.832,E2 -12440.832} C_VEL
LIN {X 0,Y 375.985,Z 235.151,A -85,B 0,C 180,E1 -12444.281,E2 -12444.281} C_VEL
LIN {X 0,Y 376.017,Z 235.126,A -85,B 0,C 180,E1 -12446.652,E2 -12446.652} C_VEL
LIN {X 0,Y 375.961,Z 235.155,A -85,B 0,C 180,E1 -12450.312,E2 -12450.312} C_VEL
LIN {X 0,Y 375.957,Z 235.14,A -85,B 0,C 180,E1 -12454.111,E2 -12454.111} C_VEL
LIN {X 0,Y 375.952,Z 235.154,A -85,B 0,C 180,E1 -12456.741,E2 -12456.741} C_VEL
LIN {X 0,Y 375.992,Z 235.14,A -85,B 0,C 180,E1 -12459.972,E2 -12459.972} C_VEL
LIN {X 0,Y 375.986,Z 235.149,A -85,B 0,C 180,E1 -12463.198,E2 -12463.198} C_VEL
LIN {X 0,Y 375.933,Z 235.128,A -85,B 0,C 180,E1 -12466.81,E2 -12466.81} C_VEL
LIN {X 0,Y 375.994,Z 235.133,A -85,B 0,C 180,E1 -12470.027,E2 -12470.027} C_VEL
LIN {X 0,Y 375.961,Z 235.145,A -85,B 0,C 180,E1 -12473.495,E2 -12473.495} C_VEL
LIN {X 0,Y 375.956,Z 235.131,A -85,B 0,C 180,E1 -12475.888,E2 -12475.888} C_VEL
LIN {X 0,Y 375.961,Z 235.141,A -85,B 0,C 180,E1 -12479.687,E2 -12479.687} C_VEL
LIN {X 0,Y 376.016,Z 235.149,A -85,B 0,C 180,E1 -12483.348,E2 -12483.348} C_VEL
LIN {X 0,Y 375.993,Z 235.152,A -85,B 0,C 180,E1 -12486.888,E2 -12486.888} C_VEL
LIN {X 0,Y 375.994,Z 235.151,A -85,B 0,C 180,E1 -12490.339,E2 -12490.339} C_VEL
LIN {X 0,Y 376.025,Z 235.149,A -85,B 0,C 180,E1 -12493.719,E2 -12493.719} C_VEL
LIN {X 0,Y 376.115,Z 235.391,A -85,B 0,C 180,E1 -12496.076,E2 -12496.076} C_VEL
LIN {X 0,Y 376.404,Z 236.521,A -85,B 0,C 180,E1 -12496.466,E2 -12496.466} C_VEL
LIN {X 0,Y 377.861,Z 239.024,A -85,B 0,C 180,E1 -12497.103,E2 -12497.103} C_VEL
LIN {X 0,Y 380.042,Z 240.683,A -85,B 0,C 180,E1 -12497.945,E2 -12497.945} C_VEL
LIN {X 0,Y 381.205,Z 241.43,A -85,B 0,C 180,E1 -12498.434,E2 -12498.434} C_VEL
LIN {X 0,Y 382.608,Z 243.819,A -85,B 0,C 180,E1 -12499.081,E2 -12499.081} C_VEL
LIN {X 0,Y 384.915,Z 246.149,A -85,B 0,C 180,E1 -12500.234,E2 -12500.234} C_VEL
LIN {X 0,Y 387.591,Z 247.679,A -85,B 0,C 180,E1 -12501.659,E2 -12501.659} C_VEL
LIN {X 0,Y 389.285,Z 250.434,A -85,B 0,C 180,E1 -12502.841,E2 -12502.841} C_VEL
LIN {X 0,Y 391.041,Z 252.139,A -85,B 0,C 180,E1 -12504.198,E2 -12504.198} C_VEL
LIN {X 0,Y 392.756,Z 253.217,A -85,B 0,C 180,E1 -12505.895,E2 -12505.895} C_VEL
LIN {X 0,Y 393.915,Z 253.583,A -85,B 0,C 180,E1 -12507.576,E2 -12507.576} C_VEL
LIN {X 0,Y 394.407,Z 254.003,A -85,B 0,C 180,E1 -12508.979,E2 -12508.979} C_VEL
LIN {X 0,Y 394.593,Z 253.943,A -85,B 0,C 180,E1 -12510,E2 -12510} C_VEL
LIN {X 0,Y 394.096,Z 253.716,A -85,B 0,C 180,E1 -12512.044,E2 -12512.044} C_VEL
LIN {X 0,Y 393.066,Z 253.319,A -85,B 0,C 180,E1 -12513.725,E2 -12513.725} C_VEL
LIN {X 0,Y 391.609,Z 252.582,A -85,B 0,C 180,E1 -12515.277,E2 -12515.277} C_VEL
LIN {X 0,Y 389.867,Z 251.111,A -85,B 0,C 180,E1 -12516.729,E2 -12516.729} C_VEL
LIN {X 0,Y 388.033,Z 248.48,A -85,B 0,C 180,E1 -12518.061,E2 -12518.061} C_VEL
LIN {X 0,Y 387.368,Z 247.385,A -85,B 0,C 180,E1 -12518.477,E2 -12518.477} C_VEL
LIN {X 0,Y 384.676,Z 245.97,A -85,B 0,C 180,E1 -12519.881,E2 -12519.881} C_VEL
LIN {X 0,Y 382.443,Z 243.627,A -85,B 0,C 180,E1 -12520.991,E2 -12520.991} C_VEL
LIN {X 0,Y 380.868,Z 241.114,A -85,B 0,C 180,E1 -12521.711,E2 -12521.711} C_VEL
LIN {X 0,Y 378.262,Z 239.429,A -85,B 0,C 180,E1 -12522.746,E2 -12522.746} C_VEL
LIN {X 0,Y 376.574,Z 236.984,A -85,B 0,C 180,E1 -12523.445,E2 -12523.445} C_VEL
LIN {X 0,Y 376.2,Z 235.745,A -85,B 0,C 180,E1 -12523.73,E2 -12523.73} C_VEL
LIN {X 0,Y 376.064,Z 235.165,A -85,B 0,C 180,E1 -12524.337,E2 -12524.337} C_VEL
LIN {X 0,Y 376.04,Z 235.146,A -85,B 0,C 180,E1 -12527.608,E2 -12527.608} C_VEL
LIN {X 0,Y 375.974,Z 235.154,A -85,B 0,C 180,E1 -12530.832,E2 -12530.832} C_VEL
LIN {X 0,Y 375.99,Z 235.152,A -85,B 0,C 180,E1 -12534.282,E2 -12534.282} C_VEL
LIN {X 0,Y 376.016,Z 235.149,A -85,B 0,C 180,E1 -12536.652,E2 -12536.652} C_VEL
LIN {X 0,Y 375.961,Z 235.14,A -85,B 0,C 180,E1 -12540.313,E2 -12540.313} C_VEL
LIN {X 0,Y 375.956,Z 235.131,A -85,B 0,C 180,E1 -12544.112,E2 -12544.112} C_VEL
LIN {X 0,Y 375.951,Z 235.151,A -85,B 0,C 180,E1 -12546.741,E2 -12546.741} C_VEL
LIN {X 0,Y 375.989,Z 235.133,A -85,B 0,C 180,E1 -12550.031,E2 -12550.031} C_VEL
LIN {X 0,Y 375.272,Z 235.21,A -85,B 0,C 180,E1 -12550.924,E2 -12550.924} C_VEL
LIN {X 0,Y 372.363,Z 235.564,A -85,B 0,C 180,E1 -12552.376,E2 -12552.376} C_VEL
LIN {X 0,Y 369.957,Z 235.876,A -85,B 0,C 180,E1 -12553.55,E2 -12553.55} C_VEL
LIN {X 0,Y 368.972,Z 236.01,A -85,B 0,C 180,E1 -12554.459,E2 -12554.459} C_VEL
LIN {X 0,Y 368.916,Z 236.023,A -85,B 0,C 180,E1 -12554.766,E2 -12554.766} C_VEL
LIN {X 0,Y 368.942,Z 236.02,A -85,B 0,C 180,E1 -12558.187,E2 -12558.187} C_VEL
LIN {X 0,Y 368.909,Z 236.029,A -85,B 0,C 180,E1 -12561.359,E2 -12561.359} C_VEL
LIN {X 0,Y 368.934,Z 236.014,A -85,B 0,C 180,E1 -12565.147,E2 -12565.147} C_VEL
LIN {X 0,Y 368.926,Z 236.029,A -85,B 0,C 180,E1 -12569.047,E2 -12569.047} C_VEL
LIN {X 0,Y 368.973,Z 236.009,A -85,B 0,C 180,E1 -12571.564,E2 -12571.564} C_VEL
LIN {X 0,Y 368.997,Z 236.009,A -85,B 0,C 180,E1 -12574.02,E2 -12574.02} C_VEL
LIN {X 0,Y 368.92,Z 236.03,A -85,B 0,C 180,E1 -12577.605,E2 -12577.605} C_VEL
LIN {X 0,Y 368.956,Z 236,A -85,B 0,C 180,E1 -12581.106,E2 -12581.106} C_VEL
LIN {X 0,Y 368.996,Z 236.018,A -85,B 0,C 180,E1 -12584.536,E2 -12584.536} C_VEL
LIN {X 0,Y 369.003,Z 236.007,A -85,B 0,C 180,E1 -12587.907,E2 -12587.907} C_VEL
LIN {X 0,Y 369.164,Z 235.987,A -85,B 0,C 180,E1 -12591.87,E2 -12591.87} C_VEL
LIN {X 0,Y 369.141,Z 236.001,A -85,B 0,C 180,E1 -12594.538,E2 -12594.538} C_VEL
LIN {X 0,Y 369.317,Z 235.965,A -85,B 0,C 180,E1 -12597.819,E2 -12597.819} C_VEL
LIN {X 0,Y 369.456,Z 235.934,A -85,B 0,C 180,E1 -12600.001,E2 -12600.001} C_VEL
LIN {X 0,Y 369.316,Z 235.971,A -85,B 0,C 180,E1 -12602.182,E2 -12602.182} C_VEL
LIN {X 0,Y 369.173,Z 235.996,A -85,B 0,C 180,E1 -12606.559,E2 -12606.559} C_VEL
LIN {X 0,Y 369.063,Z 235.983,A -85,B 0,C 180,E1 -12609.869,E2 -12609.869} C_VEL
LIN {X 0,Y 369.037,Z 236.012,A -85,B 0,C 180,E1 -12613.773,E2 -12613.773} C_VEL
LIN {X 0,Y 368.991,Z 235.999,A -85,B 0,C 180,E1 -12617.743,E2 -12617.743} C_VEL
LIN {X 0,Y 368.928,Z 236.025,A -85,B 0,C 180,E1 -12621.22,E2 -12621.22} C_VEL
LIN {X 0,Y 368.956,Z 236.017,A -85,B 0,C 180,E1 -12624.776,E2 -12624.776} C_VEL
LIN {X 0,Y 368.964,Z 236.005,A -85,B 0,C 180,E1 -12627.204,E2 -12627.204} C_VEL
LIN {X 0,Y 368.93,Z 236.029,A -85,B 0,C 180,E1 -12630.954,E2 -12630.954} C_VEL
LIN {X 0,Y 368.924,Z 236.019,A -85,B 0,C 180,E1 -12635.001,E2 -12635.001} C_VEL
LIN {X 0,Y 368.908,Z 236.027,A -85,B 0,C 180,E1 -12638.64,E2 -12638.64} C_VEL
LIN {X 0,Y 368.883,Z 236.034,A -85,B 0,C 180,E1 -12642.01,E2 -12642.01} C_VEL
LIN {X 0,Y 368.881,Z 236.032,A -85,B 0,C 180,E1 -12645.176,E2 -12645.176} C_VEL
LIN {X 0,Y 368.884,Z 236.023,A -85,B 0,C 180,E1 -12648.178,E2 -12648.178} C_VEL
LIN {X 0,Y 368.911,Z 236.028,A -85,B 0,C 180,E1 -12651.36,E2 -12651.36} C_VEL
LIN {X 0,Y 368.939,Z 236.019,A -85,B 0,C 180,E1 -12655.147,E2 -12655.147} C_VEL
LIN {X 0,Y 368.958,Z 236.196,A -85,B 0,C 180,E1 -12658.76,E2 -12658.76} C_VEL
LIN {X 0,Y 370.714,Z 244.933,A -85,B 0,C 180,E1 -12661.709,E2 -12661.709} C_VEL
LIN {X 0,Y 371.904,Z 252.246,A -85,B 0,C 180,E1 -12663.937,E2 -12663.937} C_VEL
LIN {X 0,Y 371.356,Z 259.378,A -85,B 0,C 180,E1 -12665.99,E2 -12665.99} C_VEL
LIN {X 0,Y 370.59,Z 267.23,A -85,B 0,C 180,E1 -12668.27,E2 -12668.27} C_VEL
LIN {X 0,Y 371.475,Z 271.898,A -85,B 0,C 180,E1 -12668.474,E2 -12668.474} C_VEL
LIN {X 0,Y 376.778,Z 300.567,A -85,B 0,C 180,E1 -12669.361,E2 -12669.361} C_VEL
LIN {X 0,Y 375.679,Z 372.093,A -85,B 0,C 180,E1 -12670.748,E2 -12670.748} C_VEL
LIN {X 0,Y 375.295,Z 381.989,A -85,B 0,C 180,E1 -12671.047,E2 -12671.047} C_VEL
LIN {X 0,Y 374.7,Z 391.964,A -85,B 0,C 180,E1 -12671.477,E2 -12671.477} C_VEL
LIN {X 0,Y 374.024,Z 401.318,A -85,B 0,C 180,E1 -12672.009,E2 -12672.009} C_VEL
LIN {X 0,Y 373.23,Z 411.46,A -85,B 0,C 180,E1 -12672.748,E2 -12672.748} C_VEL
LIN {X 0,Y 372.377,Z 420.456,A -85,B 0,C 180,E1 -12673.555,E2 -12673.555} C_VEL
LIN {X 0,Y 371.519,Z 429.184,A -85,B 0,C 180,E1 -12674.502,E2 -12674.502} C_VEL
LIN {X 0,Y 370.777,Z 436.793,A -85,B 0,C 180,E1 -12675.485,E2 -12675.485} C_VEL
LIN {X 0,Y 370.088,Z 443.801,A -85,B 0,C 180,E1 -12676.548,E2 -12676.548} C_VEL
LIN {X 0,Y 369.408,Z 450.003,A -85,B 0,C 180,E1 -12677.641,E2 -12677.641} C_VEL
LIN {X 0,Y 368.694,Z 456.539,A -85,B 0,C 180,E1 -12679.011,E2 -12679.011} C_VEL
LIN {X 0,Y 368.289,Z 461.042,A -85,B 0,C 180,E1 -12680.111,E2 -12680.111} C_VEL
LIN {X 0,Y 367.841,Z 466.534,A -85,B 0,C 180,E1 -12681.761,E2 -12681.761} C_VEL
LIN {X 0,Y 367.565,Z 470.859,A -85,B 0,C 180,E1 -12683.412,E2 -12683.412} C_VEL
LIN {X 0,Y 367.465,Z 473.226,A -85,B 0,C 180,E1 -12684.513,E2 -12684.513} C_VEL
LIN {X 0,Y 367.437,Z 475.025,A -85,B 0,C 180,E1 -12685.612,E2 -12685.612} C_VEL
LIN {X 0,Y 367.36,Z 477.469,A -85,B 0,C 180,E1 -12687.807,E2 -12687.807} C_VEL
LIN {X 0,Y 367.403,Z 478.059,A -85,B 0,C 180,E1 -12688.904,E2 -12688.904} C_VEL
LIN {X 0,Y 367.403,Z 478.059,A -85,B 0,C 180,E1 -12691.096,E2 -12691.096} C_VEL
LIN {X 0,Y 367.36,Z 477.469,A -85,B 0,C 180,E1 -12692.193,E2 -12692.193} C_VEL
LIN {X 0,Y 367.437,Z 475.025,A -85,B 0,C 180,E1 -12694.388,E2 -12694.388} C_VEL
LIN {X 0,Y 367.48,Z 472.133,A -85,B 0,C 180,E1 -12696.012,E2 -12696.012} C_VEL
LIN {X 0,Y 367.718,Z 468.087,A -85,B 0,C 180,E1 -12697.688,E2 -12697.688} C_VEL
LIN {X 0,Y 368.112,Z 462.957,A -85,B 0,C 180,E1 -12699.339,E2 -12699.339} C_VEL
LIN {X 0,Y 368.608,Z 457.695,A -85,B 0,C 180,E1 -12700.713,E2 -12700.713} C_VEL
LIN {X 0,Y 369.237,Z 451.378,A -85,B 0,C 180,E1 -12702.086,E2 -12702.086} C_VEL
LIN {X 0,Y 369.889,Z 445.428,A -85,B 0,C 180,E1 -12703.18,E2 -12703.18} C_VEL
LIN {X 0,Y 370.575,Z 438.499,A -85,B 0,C 180,E1 -12704.273,E2 -12704.273} C_VEL
LIN {X 0,Y 371.392,Z 430.319,A -85,B 0,C 180,E1 -12705.363,E2 -12705.363} C_VEL
LIN {X 0,Y 372.227,Z 421.807,A -85,B 0,C 180,E1 -12706.311,E2 -12706.311} C_VEL
LIN {X 0,Y 373.051,Z 413.091,A -85,B 0,C 180,E1 -12707.119,E2 -12707.119} C_VEL
LIN {X 0,Y 373.882,Z 403.333,A -85,B 0,C 180,E1 -12707.856,E2 -12707.856} C_VEL
LIN {X 0,Y 374.609,Z 393.251,A -85,B 0,C 180,E1 -12708.457,E2 -12708.457} C_VEL
LIN {X 0,Y 375.209,Z 383.738,A -85,B 0,C 180,E1 -12708.886,E2 -12708.886} C_VEL
LIN {X 0,Y 375.683,Z 373.426,A -85,B 0,C 180,E1 -12709.216,E2 -12709.216} C_VEL
LIN {X 0,Y 376.68,Z 300.141,A -85,B 0,C 180,E1 -12710.653,E2 -12710.653} C_VEL
LIN {X 0,Y 371.374,Z 271.35,A -85,B 0,C 180,E1 -12711.543,E2 -12711.543} C_VEL
LIN {X 0,Y 370.57,Z 267.294,A -85,B 0,C 180,E1 -12711.72,E2 -12711.72} C_VEL
LIN {X 0,Y 371.802,Z 255.3,A -85,B 0,C 180,E1 -12715.207,E2 -12715.207} C_VEL
LIN {X 0,Y 371.88,Z 251.413,A -85,B 0,C 180,E1 -12716.367,E2 -12716.367} C_VEL
LIN {X 0,Y 370.246,Z 242.483,A -85,B 0,C 180,E1 -12719.17,E2 -12719.17} C_VEL
LIN {X 0,Y 368.941,Z 236.047,A -85,B 0,C 180,E1 -12721.33,E2 -12721.33} C_VEL
LIN {X 0,Y 368.931,Z 236.019,A -85,B 0,C 180,E1 -12725.001,E2 -12725.001} C_VEL
LIN {X 0,Y 368.911,Z 236.028,A -85,B 0,C 180,E1 -12728.64,E2 -12728.64} C_VEL
LIN {X 0,Y 368.883,Z 236.025,A -85,B 0,C 180,E1 -12732.009,E2 -12732.009} C_VEL
LIN {X 0,Y 368.881,Z 236.03,A -85,B 0,C 180,E1 -12735.175,E2 -12735.175} C_VEL
LIN {X 0,Y 368.884,Z 236.033,A -85,B 0,C 180,E1 -12738.177,E2 -12738.177} C_VEL
LIN {X 0,Y 368.908,Z 236.027,A -85,B 0,C 180,E1 -12741.36,E2 -12741.36} C_VEL
LIN {X 0,Y 368.931,Z 236.017,A -85,B 0,C 180,E1 -12745.145,E2 -12745.145} C_VEL
LIN {X 0,Y 368.93,Z 236.029,A -85,B 0,C 180,E1 -12749.046,E2 -12749.046} C_VEL
LIN {X 0,Y 368.964,Z 236.005,A -85,B 0,C 180,E1 -12752.796,E2 -12752.796} C_VEL
LIN {X 0,Y 368.938,Z 236.024,A -85,B 0,C 180,E1 -12756.115,E2 -12756.115} C_VEL
LIN {X 0,Y 368.936,Z 236.011,A -85,B 0,C 180,E1 -12759.946,E2 -12759.946} C_VEL
LIN {X 0,Y 368.969,Z 236.013,A -85,B 0,C 180,E1 -12763.398,E2 -12763.398} C_VEL
LIN {X 0,Y 369.058,Z 236.012,A -85,B 0,C 180,E1 -12766.79,E2 -12766.79} C_VEL
LIN {X 0,Y 369.063,Z 235.983,A -85,B 0,C 180,E1 -12770.131,E2 -12770.131} C_VEL
LIN {X 0,Y 369.173,Z 235.996,A -85,B 0,C 180,E1 -12773.441,E2 -12773.441} C_VEL
LIN {X 0,Y 369.316,Z 235.971,A -85,B 0,C 180,E1 -12777.818,E2 -12777.818} C_VEL
LIN {X 0,Y 369.456,Z 235.934,A -85,B 0,C 180,E1 -12779.999,E2 -12779.999} C_VEL
LIN {X 0,Y 369.317,Z 235.965,A -85,B 0,C 180,E1 -12782.181,E2 -12782.181} C_VEL
LIN {X 0,Y 369.197,Z 235.994,A -85,B 0,C 180,E1 -12786.558,E2 -12786.558} C_VEL
LIN {X 0,Y 369.066,Z 235.983,A -85,B 0,C 180,E1 -12789.868,E2 -12789.868} C_VEL
LIN {X 0,Y 369.035,Z 236.013,A -85,B 0,C 180,E1 -12793.772,E2 -12793.772} C_VEL
LIN {X 0,Y 368.999,Z 236.007,A -85,B 0,C 180,E1 -12797.768,E2 -12797.768} C_VEL
LIN {X 0,Y 368.907,Z 236.024,A -85,B 0,C 180,E1 -12801.22,E2 -12801.22} C_VEL
LIN {X 0,Y 368.952,Z 236.021,A -85,B 0,C 180,E1 -12804.775,E2 -12804.775} C_VEL
LIN {X 0,Y 368.96,Z 236.002,A -85,B 0,C 180,E1 -12807.203,E2 -12807.203} C_VEL
LIN {X 0,Y 368.916,Z 236.026,A -85,B 0,C 180,E1 -12809.689,E2 -12809.689} C_VEL
LIN {X 0,Y 368.894,Z 236.026,A -85,B 0,C 180,E1 -12813.043,E2 -12813.043} C_VEL
LIN {X 0,Y 368.915,Z 236.026,A -85,B 0,C 180,E1 -12816.196,E2 -12816.196} C_VEL
LIN {X 0,Y 368.903,Z 236.029,A -85,B 0,C 180,E1 -12818.952,E2 -12818.952} C_VEL
LIN {X 0,Y 368.947,Z 236.022,A -85,B 0,C 180,E1 -12822.021,E2 -12822.021} C_VEL
LIN {X 0,Y 368.921,Z 236.024,A -85,B 0,C 180,E1 -12825.182,E2 -12825.182} C_VEL
LIN {X 0,Y 368.89,Z 235.995,A -85,B 0,C 180,E1 -12828.179,E2 -12828.179} C_VEL
LIN {X 0,Y 368.909,Z 236.03,A -85,B 0,C 180,E1 -12831.359,E2 -12831.359} C_VEL
LIN {X 0,Y 368.933,Z 236.004,A -85,B 0,C 180,E1 -12835.146,E2 -12835.146} C_VEL
LIN {X 0,Y 368.925,Z 236.028,A -85,B 0,C 180,E1 -12839.046,E2 -12839.046} C_VEL
LIN {X 0,Y 368.959,Z 236.027,A -85,B 0,C 180,E1 -12842.796,E2 -12842.796} C_VEL
LIN {X 0,Y 368.942,Z 236.03,A -85,B 0,C 180,E1 -12846.113,E2 -12846.113} C_VEL
LIN {X 0,Y 368.933,Z 236.031,A -85,B 0,C 180,E1 -12849.947,E2 -12849.947} C_VEL
LIN {X 0,Y 368.972,Z 236.026,A -85,B 0,C 180,E1 -12853.399,E2 -12853.399} C_VEL
LIN {X 0,Y 369.037,Z 236.422,A -85,B 0,C 180,E1 -12854.112,E2 -12854.112} C_VEL
LIN {X 0,Y 369.449,Z 237.784,A -85,B 0,C 180,E1 -12854.431,E2 -12854.431} C_VEL
LIN {X 0,Y 370.843,Z 239.96,A -85,B 0,C 180,E1 -12854.93,E2 -12854.93} C_VEL
LIN {X 0,Y 373.911,Z 242.227,A -85,B 0,C 180,E1 -12855.939,E2 -12855.939} C_VEL
LIN {X 0,Y 375.802,Z 245.292,A -85,B 0,C 180,E1 -12856.694,E2 -12856.694} C_VEL
LIN {X 0,Y 378.433,Z 247.423,A -85,B 0,C 180,E1 -12857.668,E2 -12857.668} C_VEL
LIN {X 0,Y 379.535,Z 248.194,A -85,B 0,C 180,E1 -12858.132,E2 -12858.132} C_VEL
LIN {X 0,Y 381.399,Z 250.938,A -85,B 0,C 180,E1 -12858.978,E2 -12858.978} C_VEL
LIN {X 0,Y 383.705,Z 253.064,A -85,B 0,C 180,E1 -12860.095,E2 -12860.095} C_VEL
LIN {X 0,Y 386.289,Z 254.545,A -85,B 0,C 180,E1 -12861.433,E2 -12861.433} C_VEL
LIN {X 0,Y 388.224,Z 257.441,A -85,B 0,C 180,E1 -12862.72,E2 -12862.72} C_VEL
LIN {X 0,Y 390.286,Z 259.323,A -85,B 0,C 180,E1 -12864.316,E2 -12864.316} C_VEL
LIN {X 0,Y 391.884,Z 260.241,A -85,B 0,C 180,E1 -12865.886,E2 -12865.886} C_VEL
LIN {X 0,Y 392.995,Z 260.604,A -85,B 0,C 180,E1 -12867.456,E2 -12867.456} C_VEL
LIN {X 0,Y 393.545,Z 261.049,A -85,B 0,C 180,E1 -12868.977,E2 -12868.977} C_VEL
LIN {X 0,Y 393.727,Z 260.99,A -85,B 0,C 180,E1 -12870,E2 -12870} C_VEL
LIN {X 0,Y 393.467,Z 260.923,A -85,B 0,C 180,E1 -12871.535,E2 -12871.535} C_VEL
LIN {X 0,Y 392.738,Z 260.496,A -85,B 0,C 180,E1 -12873.077,E2 -12873.077} C_VEL
LIN {X 0,Y 391.175,Z 259.886,A -85,B 0,C 180,E1 -12874.896,E2 -12874.896} C_VEL
LIN {X 0,Y 389.129,Z 258.375,A -85,B 0,C 180,E1 -12876.62,E2 -12876.62} C_VEL
LIN {X 0,Y 387.407,Z 256.295,A -85,B 0,C 180,E1 -12877.871,E2 -12877.871} C_VEL
LIN {X 0,Y 385.95,Z 254.185,A -85,B 0,C 180,E1 -12878.772,E2 -12878.772} C_VEL
LIN {X 0,Y 383.231,Z 252.733,A -85,B 0,C 180,E1 -12880.134,E2 -12880.134} C_VEL
LIN {X 0,Y 380.895,Z 250.358,A -85,B 0,C 180,E1 -12881.238,E2 -12881.238} C_VEL
LIN {X 0,Y 379.161,Z 247.783,A -85,B 0,C 180,E1 -12882.036,E2 -12882.036} C_VEL
LIN {X 0,Y 376.571,Z 246.099,A -85,B 0,C 180,E1 -12883.011,E2 -12883.011} C_VEL
LIN {X 0,Y 374.518,Z 243.35,A -85,B 0,C 180,E1 -12883.833,E2 -12883.833} C_VEL
LIN {X 0,Y 373.644,Z 241.875,A -85,B 0,C 180,E1 -12884.154,E2 -12884.154} C_VEL
LIN {X 0,Y 370.852,Z 239.963,A -85,B 0,C 180,E1 -12885.068,E2 -12885.068} C_VEL
LIN {X 0,Y 369.45,Z 237.787,A -85,B 0,C 180,E1 -12885.569,E2 -12885.569} C_VEL
LIN {X 0,Y 369.037,Z 236.424,A -85,B 0,C 180,E1 -12885.888,E2 -12885.888} C_VEL
LIN {X 0,Y 368.972,Z 236.026,A -85,B 0,C 180,E1 -12886.601,E2 -12886.601} C_VEL
LIN {X 0,Y 368.933,Z 236.031,A -85,B 0,C 180,E1 -12890.053,E2 -12890.053} C_VEL
LIN {X 0,Y 368.942,Z 236.03,A -85,B 0,C 180,E1 -12893.887,E2 -12893.887} C_VEL
LIN {X 0,Y 368.959,Z 236.027,A -85,B 0,C 180,E1 -12897.204,E2 -12897.204} C_VEL
LIN {X 0,Y 368.925,Z 236.028,A -85,B 0,C 180,E1 -12900.954,E2 -12900.954} C_VEL
LIN {X 0,Y 368.925,Z 236.005,A -85,B 0,C 180,E1 -12905.002,E2 -12905.002} C_VEL
LIN {X 0,Y 368.909,Z 236.03,A -85,B 0,C 180,E1 -12908.641,E2 -12908.641} C_VEL
LIN {X 0,Y 368.89,Z 235.995,A -85,B 0,C 180,E1 -12911.821,E2 -12911.821} C_VEL
LIN {X 0,Y 368.916,Z 236.023,A -85,B 0,C 180,E1 -12914.766,E2 -12914.766} C_VEL
LIN {X 0,Y 368.315,Z 236.111,A -85,B 0,C 180,E1 -12915.677,E2 -12915.677} C_VEL
LIN {X 0,Y 365.487,Z 236.46,A -85,B 0,C 180,E1 -12917.159,E2 -12917.159} C_VEL
LIN {X 0,Y 363.041,Z 236.753,A -85,B 0,C 180,E1 -12918.357,E2 -12918.357} C_VEL
LIN {X 0,Y 361.975,Z 236.882,A -85,B 0,C 180,E1 -12919.284,E2 -12919.284} C_VEL
LIN {X 0,Y 361.881,Z 236.894,A -85,B 0,C 180,E1 -12919.598,E2 -12919.598} C_VEL
LIN {X 0,Y 361.866,Z 236.908,A -85,B 0,C 180,E1 -12922.983,E2 -12922.983} C_VEL
LIN {X 0,Y 361.855,Z 236.903,A -85,B 0,C 180,E1 -12926.631,E2 -12926.631} C_VEL
LIN {X 0,Y 361.872,Z 236.91,A -85,B 0,C 180,E1 -12929.673,E2 -12929.673} C_VEL
LIN {X 0,Y 361.951,Z 236.878,A -85,B 0,C 180,E1 -12933.476,E2 -12933.476} C_VEL
LIN {X 0,Y 361.877,Z 236.908,A -85,B 0,C 180,E1 -12937.145,E2 -12937.145} C_VEL
LIN {X 0,Y 361.904,Z 236.878,A -85,B 0,C 180,E1 -12940.724,E2 -12940.724} C_VEL
LIN {X 0,Y 361.931,Z 236.89,A -85,B 0,C 180,E1 -12943.067,E2 -12943.067} C_VEL
LIN {X 0,Y 361.997,Z 236.889,A -85,B 0,C 180,E1 -12946.528,E2 -12946.528} C_VEL
LIN {X 0,Y 362.03,Z 236.858,A -85,B 0,C 180,E1 -12949.939,E2 -12949.939} C_VEL
LIN {X 0,Y 362.159,Z 236.868,A -85,B 0,C 180,E1 -12953.314,E2 -12953.314} C_VEL
LIN {X 0,Y 362.281,Z 236.841,A -85,B 0,C 180,E1 -12957.777,E2 -12957.777} C_VEL
LIN {X 0,Y 362.425,Z 236.809,A -85,B 0,C 180,E1 -12960.001,E2 -12960.001} C_VEL
LIN {X 0,Y 362.28,Z 236.847,A -85,B 0,C 180,E1 -12962.224,E2 -12962.224} C_VEL
LIN {X 0,Y 362.135,Z 236.871,A -85,B 0,C 180,E1 -12966.687,E2 -12966.687} C_VEL
LIN {X 0,Y 362,Z 236.863,A -85,B 0,C 180,E1 -12970.064,E2 -12970.064} C_VEL
LIN {X 0,Y 361.998,Z 236.888,A -85,B 0,C 180,E1 -12973.899,E2 -12973.899} C_VEL
LIN {X 0,Y 361.928,Z 236.884,A -85,B 0,C 180,E1 -12976.935,E2 -12976.935} C_VEL
LIN {X 0,Y 361.887,Z 236.891,A -85,B 0,C 180,E1 -12980.461,E2 -12980.461} C_VEL
LIN {X 0,Y 361.894,Z 236.902,A -85,B 0,C 180,E1 -12984.113,E2 -12984.113} C_VEL
LIN {X 0,Y 361.942,Z 236.878,A -85,B 0,C 180,E1 -12986.722,E2 -12986.722} C_VEL
LIN {X 0,Y 361.874,Z 236.908,A -85,B 0,C 180,E1 -12990.329,E2 -12990.329} C_VEL
LIN {X 0,Y 361.851,Z 236.894,A -85,B 0,C 180,E1 -12994.281,E2 -12994.281} C_VEL
LIN {X 0,Y 361.862,Z 236.908,A -85,B 0,C 180,E1 -12997.223,E2 -12997.223} C_VEL
LIN {X 0,Y 361.836,Z 236.906,A -85,B 0,C 180,E1 -13000.756,E2 -13000.756} C_VEL
LIN {X 0,Y 361.818,Z 236.909,A -85,B 0,C 180,E1 -13004.369,E2 -13004.369} C_VEL
LIN {X 0,Y 361.838,Z 236.911,A -85,B 0,C 180,E1 -13007.569,E2 -13007.569} C_VEL
LIN {X 0,Y 361.872,Z 236.898,A -85,B 0,C 180,E1 -13010.974,E2 -13010.974} C_VEL
LIN {X 0,Y 361.876,Z 236.895,A -85,B 0,C 180,E1 -13014.656,E2 -13014.656} C_VEL
LIN {X 0,Y 361.913,Z 237.004,A -85,B 0,C 180,E1 -13018.378,E2 -13018.378} C_VEL
LIN {X 0,Y 363.468,Z 244.747,A -85,B 0,C 180,E1 -13021.092,E2 -13021.092} C_VEL
LIN {X 0,Y 364.943,Z 253.112,A -85,B 0,C 180,E1 -13023.709,E2 -13023.709} C_VEL
LIN {X 0,Y 364.497,Z 259.187,A -85,B 0,C 180,E1 -13025.509,E2 -13025.509} C_VEL
LIN {X 0,Y 363.674,Z 267.089,A -85,B 0,C 180,E1 -13027.844,E2 -13027.844} C_VEL
LIN {X 0,Y 365.006,Z 273.7,A -85,B 0,C 180,E1 -13028.114,E2 -13028.114} C_VEL
LIN {X 0,Y 370.049,Z 300.972,A -85,B 0,C 180,E1 -13028.98,E2 -13028.98} C_VEL
LIN {X 0,Y 368.997,Z 371.9,A -85,B 0,C 180,E1 -13030.386,E2 -13030.386} C_VEL
LIN {X 0,Y 368.595,Z 381.797,A -85,B 0,C 180,E1 -13030.689,E2 -13030.689} C_VEL
LIN {X 0,Y 367.986,Z 391.771,A -85,B 0,C 180,E1 -13031.126,E2 -13031.126} C_VEL
LIN {X 0,Y 367.193,Z 402.133,A -85,B 0,C 180,E1 -13031.735,E2 -13031.735} C_VEL
LIN {X 0,Y 366.446,Z 411.267,A -85,B 0,C 180,E1 -13032.418,E2 -13032.418} C_VEL
LIN {X 0,Y 365.544,Z 420.262,A -85,B 0,C 180,E1 -13033.238,E2 -13033.238} C_VEL
LIN {X 0,Y 364.646,Z 428.99,A -85,B 0,C 180,E1 -13034.203,E2 -13034.203} C_VEL
LIN {X 0,Y 363.846,Z 436.964,A -85,B 0,C 180,E1 -13035.257,E2 -13035.257} C_VEL
LIN {X 0,Y 362.944,Z 445.234,A -85,B 0,C 180,E1 -13036.564,E2 -13036.564} C_VEL
LIN {X 0,Y 362.26,Z 451.184,A -85,B 0,C 180,E1 -13037.678,E2 -13037.678} C_VEL
LIN {X 0,Y 361.587,Z 457.501,A -85,B 0,C 180,E1 -13039.076,E2 -13039.076} C_VEL
LIN {X 0,Y 361.065,Z 462.763,A -85,B 0,C 180,E1 -13040.477,E2 -13040.477} C_VEL
LIN {X 0,Y 360.669,Z 467.894,A -85,B 0,C 180,E1 -13042.16,E2 -13042.16} C_VEL
LIN {X 0,Y 360.5,Z 470.665,A -85,B 0,C 180,E1 -13043.283,E2 -13043.283} C_VEL
LIN {X 0,Y 360.385,Z 473.033,A -85,B 0,C 180,E1 -13044.404,E2 -13044.404} C_VEL
LIN {X 0,Y 360.349,Z 474.832,A -85,B 0,C 180,E1 -13045.526,E2 -13045.526} C_VEL
LIN {X 0,Y 360.264,Z 477.276,A -85,B 0,C 180,E1 -13047.764,E2 -13047.764} C_VEL
LIN {X 0,Y 360.303,Z 477.866,A -85,B 0,C 180,E1 -13048.882,E2 -13048.882} C_VEL
LIN {X 0,Y 360.303,Z 477.866,A -85,B 0,C 180,E1 -13051.118,E2 -13051.118} C_VEL
LIN {X 0,Y 360.264,Z 477.276,A -85,B 0,C 180,E1 -13052.236,E2 -13052.236} C_VEL
LIN {X 0,Y 360.349,Z 474.832,A -85,B 0,C 180,E1 -13054.474,E2 -13054.474} C_VEL
LIN {X 0,Y 360.379,Z 472.307,A -85,B 0,C 180,E1 -13055.961,E2 -13055.961} C_VEL
LIN {X 0,Y 360.592,Z 469.425,A -85,B 0,C 180,E1 -13057.278,E2 -13057.278} C_VEL
LIN {X 0,Y 360.921,Z 464.68,A -85,B 0,C 180,E1 -13058.962,E2 -13058.962} C_VEL
LIN {X 0,Y 361.506,Z 458.658,A -85,B 0,C 180,E1 -13060.643,E2 -13060.643} C_VEL
LIN {X 0,Y 362.092,Z 452.56,A -85,B 0,C 180,E1 -13062.043,E2 -13062.043} C_VEL
LIN {X 0,Y 362.771,Z 446.861,A -85,B 0,C 180,E1 -13063.158,E2 -13063.158} C_VEL
LIN {X 0,Y 363.684,Z 438.306,A -85,B 0,C 180,E1 -13064.55,E2 -13064.55} C_VEL
LIN {X 0,Y 364.527,Z 430.125,A -85,B 0,C 180,E1 -13065.659,E2 -13065.659} C_VEL
LIN {X 0,Y 365.409,Z 421.614,A -85,B 0,C 180,E1 -13066.624,E2 -13066.624} C_VEL
LIN {X 0,Y 366.275,Z 412.898,A -85,B 0,C 180,E1 -13067.446,E2 -13067.446} C_VEL
LIN {X 0,Y 367.095,Z 403.139,A -85,B 0,C 180,E1 -13068.198,E2 -13068.198} C_VEL
LIN {X 0,Y 367.886,Z 393.059,A -85,B 0,C 180,E1 -13068.807,E2 -13068.807} C_VEL
LIN {X 0,Y 368.522,Z 383.546,A -85,B 0,C 180,E1 -13069.242,E2 -13069.242} C_VEL
LIN {X 0,Y 368.976,Z 373.233,A -85,B 0,C 180,E1 -13069.579,E2 -13069.579} C_VEL
LIN {X 0,Y 370.173,Z 302.609,A -85,B 0,C 180,E1 -13070.979,E2 -13070.979} C_VEL
LIN {X 0,Y 366.398,Z 280.369,A -85,B 0,C 180,E1 -13071.661,E2 -13071.661} C_VEL
LIN {X 0,Y 363.694,Z 267.361,A -85,B 0,C 180,E1 -13072.126,E2 -13072.126} C_VEL
LIN {X 0,Y 363.679,Z 266.649,A -85,B 0,C 180,E1 -13072.239,E2 -13072.239} C_VEL
LIN {X 0,Y 364.965,Z 255.242,A -85,B 0,C 180,E1 -13075.675,E2 -13075.675} C_VEL
LIN {X 0,Y 364.739,Z 251.368,A -85,B 0,C 180,E1 -13076.878,E2 -13076.878} C_VEL
LIN {X 0,Y 363.031,Z 242.43,A -85,B 0,C 180,E1 -13079.767,E2 -13079.767} C_VEL
LIN {X 0,Y 361.902,Z 236.93,A -85,B 0,C 180,E1 -13081.664,E2 -13081.664} C_VEL
LIN {X 0,Y 361.87,Z 236.895,A -85,B 0,C 180,E1 -13085.636,E2 -13085.636} C_VEL
LIN {X 0,Y 361.872,Z 236.898,A -85,B 0,C 180,E1 -13089.026,E2 -13089.026} C_VEL
LIN {X 0,Y 361.838,Z 236.91,A -85,B 0,C 180,E1 -13092.828,E2 -13092.828} C_VEL
LIN {X 0,Y 361.819,Z 236.91,A -85,B 0,C 180,E1 -13095.946,E2 -13095.946} C_VEL
LIN {X 0,Y 361.836,Z 236.906,A -85,B 0,C 180,E1 -13099.244,E2 -13099.244} C_VEL
LIN {X 0,Y 361.862,Z 236.908,A -85,B 0,C 180,E1 -13102.777,E2 -13102.777} C_VEL
LIN {X 0,Y 361.851,Z 236.894,A -85,B 0,C 180,E1 -13105.719,E2 -13105.719} C_VEL
LIN {X 0,Y 361.874,Z 236.908,A -85,B 0,C 180,E1 -13109.671,E2 -13109.671} C_VEL
LIN {X 0,Y 361.954,Z 236.877,A -85,B 0,C 180,E1 -13113.475,E2 -13113.475} C_VEL
LIN {X 0,Y 361.883,Z 236.908,A -85,B 0,C 180,E1 -13117.144,E2 -13117.144} C_VEL
LIN {X 0,Y 361.886,Z 236.883,A -85,B 0,C 180,E1 -13120.722,E2 -13120.722} C_VEL
LIN {X 0,Y 361.943,Z 236.891,A -85,B 0,C 180,E1 -13124.225,E2 -13124.225} C_VEL
LIN {X 0,Y 361.999,Z 236.89,A -85,B 0,C 180,E1 -13126.527,E2 -13126.527} C_VEL
LIN {X 0,Y 362,Z 236.863,A -85,B 0,C 180,E1 -13129.936,E2 -13129.936} C_VEL
LIN {X 0,Y 362.135,Z 236.871,A -85,B 0,C 180,E1 -13133.313,E2 -13133.313} C_VEL
LIN {X 0,Y 362.28,Z 236.847,A -85,B 0,C 180,E1 -13137.776,E2 -13137.776} C_VEL
LIN {X 0,Y 362.425,Z 236.809,A -85,B 0,C 180,E1 -13139.999,E2 -13139.999} C_VEL
LIN {X 0,Y 362.281,Z 236.841,A -85,B 0,C 180,E1 -13142.223,E2 -13142.223} C_VEL
LIN {X 0,Y 362.159,Z 236.868,A -85,B 0,C 180,E1 -13146.686,E2 -13146.686} C_VEL
LIN {X 0,Y 362.03,Z 236.858,A -85,B 0,C 180,E1 -13150.061,E2 -13150.061} C_VEL
LIN {X 0,Y 361.996,Z 236.89,A -85,B 0,C 180,E1 -13153.898,E2 -13153.898} C_VEL
LIN {X 0,Y 361.965,Z 236.879,A -85,B 0,C 180,E1 -13157.938,E2 -13157.938} C_VEL
LIN {X 0,Y 361.859,Z 236.903,A -85,B 0,C 180,E1 -13161.654,E2 -13161.654} C_VEL
LIN {X 0,Y 361.924,Z 236.895,A -85,B 0,C 180,E1 -13165.29,E2 -13165.29} C_VEL
LIN {X 0,Y 361.911,Z 236.881,A -85,B 0,C 180,E1 -13167.778,E2 -13167.778} C_VEL
LIN {X 0,Y 361.844,Z 236.911,A -85,B 0,C 180,E1 -13171.285,E2 -13171.285} C_VEL
LIN {X 0,Y 361.851,Z 236.895,A -85,B 0,C 180,E1 -13174.28,E2 -13174.28} C_VEL
LIN {X 0,Y 361.862,Z 236.909,A -85,B 0,C 180,E1 -13177.223,E2 -13177.223} C_VEL
LIN {X 0,Y 361.903,Z 236.891,A -85,B 0,C 180,E1 -13180.768,E2 -13180.768} C_VEL
LIN {X 0,Y 361.908,Z 236.9,A -85,B 0,C 180,E1 -13184.353,E2 -13184.353} C_VEL
LIN {X 0,Y 361.838,Z 236.872,A -85,B 0,C 180,E1 -13187.567,E2 -13187.567} C_VEL
LIN {X 0,Y 361.871,Z 236.905,A -85,B 0,C 180,E1 -13190.972,E2 -13190.972} C_VEL
LIN {X 0,Y 361.871,Z 236.886,A -85,B 0,C 180,E1 -13194.655,E2 -13194.655} C_VEL
LIN {X 0,Y 361.834,Z 236.914,A -85,B 0,C 180,E1 -13198.37,E2 -13198.37} C_VEL
LIN {X 0,Y 361.904,Z 236.901,A -85,B 0,C 180,E1 -13202.221,E2 -13202.221} C_VEL
LIN {X 0,Y 361.924,Z 236.903,A -85,B 0,C 180,E1 -13204.71,E2 -13204.71} C_VEL
LIN {X 0,Y 361.888,Z 236.908,A -85,B 0,C 180,E1 -13208.347,E2 -13208.347} C_VEL
LIN {X 0,Y 361.959,Z 237.006,A -85,B 0,C 180,E1 -13212.141,E2 -13212.141} C_VEL
LIN {X 0,Y 362.155,Z 237.987,A -85,B 0,C 180,E1 -13212.51,E2 -13212.51} C_VEL
LIN {X 0,Y 363.708,Z 240.76,A -85,B 0,C 180,E1 -13213.03,E2 -13213.03} C_VEL
LIN {X 0,Y 366.072,Z 242.534,A -85,B 0,C 180,E1 -13213.721,E2 -13213.721} C_VEL
LIN {X 0,Y 368.394,Z 245.961,A -85,B 0,C 180,E1 -13214.47,E2 -13214.47} C_VEL
LIN {X 0,Y 371.016,Z 248.151,A -85,B 0,C 180,E1 -13215.323,E2 -13215.323} C_VEL
LIN {X 0,Y 371.852,Z 248.843,A -85,B 0,C 180,E1 -13215.602,E2 -13215.602} C_VEL
LIN {X 0,Y 374.175,Z 252.038,A -85,B 0,C 180,E1 -13216.445,E2 -13216.445} C_VEL
LIN {X 0,Y 376.963,Z 254.261,A -85,B 0,C 180,E1 -13217.483,E2 -13217.483} C_VEL
LIN {X 0,Y 377.928,Z 255.054,A -85,B 0,C 180,E1 -13217.856,E2 -13217.856} C_VEL
LIN {X 0,Y 380.531,Z 258.38,A -85,B 0,C 180,E1 -13219.02,E2 -13219.02} C_VEL
LIN {X 0,Y 383.373,Z 260.504,A -85,B 0,C 180,E1 -13220.37,E2 -13220.37} C_VEL
LIN {X 0,Y 384.988,Z 261.446,A -85,B 0,C 180,E1 -13221.206,E2 -13221.206} C_VEL
LIN {X 0,Y 387.164,Z 264.427,A -85,B 0,C 180,E1 -13222.596,E2 -13222.596} C_VEL
LIN {X 0,Y 389.259,Z 266.25,A -85,B 0,C 180,E1 -13224.171,E2 -13224.171} C_VEL
LIN {X 0,Y 391.009,Z 267.286,A -85,B 0,C 180,E1 -13225.877,E2 -13225.877} C_VEL
LIN {X 0,Y 392.129,Z 267.653,A -85,B 0,C 180,E1 -13227.451,E2 -13227.451} C_VEL
LIN {X 0,Y 392.684,Z 268.085,A -85,B 0,C 180,E1 -13228.975,E2 -13228.975} C_VEL
LIN {X 0,Y 392.864,Z 268.022,A -85,B 0,C 180,E1 -13230,E2 -13230} C_VEL
LIN {X 0,Y 392.598,Z 267.971,A -85,B 0,C 180,E1 -13231.539,E2 -13231.539} C_VEL
LIN {X 0,Y 391.864,Z 267.542,A -85,B 0,C 180,E1 -13233.084,E2 -13233.084} C_VEL
LIN {X 0,Y 390.285,Z 266.931,A -85,B 0,C 180,E1 -13234.907,E2 -13234.907} C_VEL
LIN {X 0,Y 388.213,Z 265.474,A -85,B 0,C 180,E1 -13236.635,E2 -13236.635} C_VEL
LIN {X 0,Y 386.33,Z 263.397,A -85,B 0,C 180,E1 -13237.961,E2 -13237.961} C_VEL
LIN {X 0,Y 384.775,Z 261.127,A -85,B 0,C 180,E1 -13238.931,E2 -13238.931} C_VEL
LIN {X 0,Y 381.794,Z 259.488,A -85,B 0,C 180,E1 -13240.39,E2 -13240.39} C_VEL
LIN {X 0,Y 379.033,Z 256.743,A -85,B 0,C 180,E1 -13241.628,E2 -13241.628} C_VEL
LIN {X 0,Y 377.387,Z 254.465,A -85,B 0,C 180,E1 -13242.366,E2 -13242.366} C_VEL
LIN {X 0,Y 374.54,Z 252.419,A -85,B 0,C 180,E1 -13243.413,E2 -13243.413} C_VEL
LIN {X 0,Y 372.281,Z 249.506,A -85,B 0,C 180,E1 -13244.245,E2 -13244.245} C_VEL
LIN {X 0,Y 371.417,Z 248.367,A -85,B 0,C 180,E1 -13244.548,E2 -13244.548} C_VEL
LIN {X 0,Y 368.647,Z 246.259,A -85,B 0,C 180,E1 -13245.453,E2 -13245.453} C_VEL
LIN {X 0,Y 366.669,Z 243.429,A -85,B 0,C 180,E1 -13246.083,E2 -13246.083} C_VEL
LIN {X 0,Y 366.071,Z 242.534,A -85,B 0,C 180,E1 -13246.279,E2 -13246.279} C_VEL
LIN {X 0,Y 363.707,Z 240.761,A -85,B 0,C 180,E1 -13246.97,E2 -13246.97} C_VEL
LIN {X 0,Y 362.199,Z 238.117,A -85,B 0,C 180,E1 -13247.466,E2 -13247.466} C_VEL
LIN {X 0,Y 361.974,Z 237.105,A -85,B 0,C 180,E1 -13247.778,E2 -13247.778} C_VEL
LIN {X 0,Y 361.88,Z 236.91,A -85,B 0,C 180,E1 -13251.222,E2 -13251.222} C_VEL
LIN {X 0,Y 361.892,Z 236.908,A -85,B 0,C 180,E1 -13254.114,E2 -13254.114} C_VEL
LIN {X 0,Y 361.937,Z 236.903,A -85,B 0,C 180,E1 -13256.722,E2 -13256.722} C_VEL
LIN {X 0,Y 361.869,Z 236.895,A -85,B 0,C 180,E1 -13260.328,E2 -13260.328} C_VEL
LIN {X 0,Y 361.85,Z 236.886,A -85,B 0,C 180,E1 -13264.281,E2 -13264.281} C_VEL
LIN {X 0,Y 361.862,Z 236.909,A -85,B 0,C 180,E1 -13267.224,E2 -13267.224} C_VEL
LIN {X 0,Y 361.864,Z 236.88,A -85,B 0,C 180,E1 -13270.762,E2 -13270.762} C_VEL
LIN {X 0,Y 361.843,Z 236.895,A -85,B 0,C 180,E1 -13274.364,E2 -13274.364} C_VEL
LIN {X 0,Y 361.886,Z 236.907,A -85,B 0,C 180,E1 -13277.559,E2 -13277.559} C_VEL
LIN {X 0,Y 361.881,Z 236.894,A -85,B 0,C 180,E1 -13279.598,E2 -13279.598} C_VEL
LIN {X 0,Y 361.199,Z 236.988,A -85,B 0,C 180,E1 -13280.526,E2 -13280.526} C_VEL
LIN {X 0,Y 358.348,Z 237.352,A -85,B 0,C 180,E1 -13282.036,E2 -13282.036} C_VEL
LIN {X 0,Y 355.939,Z 237.647,A -85,B 0,C 180,E1 -13283.258,E2 -13283.258} C_VEL
LIN {X 0,Y 354.899,Z 237.767,A -85,B 0,C 180,E1 -13284.203,E2 -13284.203} C_VEL
LIN {X 0,Y 354.811,Z 237.775,A -85,B 0,C 180,E1 -13284.523,E2 -13284.523} C_VEL
LIN {X 0,Y 354.784,Z 237.788,A -85,B 0,C 180,E1 -13287.667,E2 -13287.667} C_VEL
LIN {X 0,Y 354.866,Z 237.774,A -85,B 0,C 180,E1 -13290.622,E2 -13290.622} C_VEL
LIN {X 0,Y 354.895,Z 237.766,A -85,B 0,C 180,E1 -13294.173,E2 -13294.173} C_VEL
LIN {X 0,Y 354.813,Z 237.783,A -85,B 0,C 180,E1 -13297.893,E2 -13297.893} C_VEL
LIN {X 0,Y 354.92,Z 237.753,A -85,B 0,C 180,E1 -13301.892,E2 -13301.892} C_VEL
LIN {X 0,Y 354.941,Z 237.77,A -85,B 0,C 180,E1 -13305.982,E2 -13305.982} C_VEL
LIN {X 0,Y 354.977,Z 237.737,A -85,B 0,C 180,E1 -13309.737,E2 -13309.737} C_VEL
LIN {X 0,Y 355.123,Z 237.743,A -85,B 0,C 180,E1 -13313.181,E2 -13313.181} C_VEL
LIN {X 0,Y 355.244,Z 237.718,A -85,B 0,C 180,E1 -13317.733,E2 -13317.733} C_VEL
LIN {X 0,Y 355.374,Z 237.686,A -85,B 0,C 180,E1 -13320.001,E2 -13320.001} C_VEL
LIN {X 0,Y 355.243,Z 237.723,A -85,B 0,C 180,E1 -13322.268,E2 -13322.268} C_VEL
LIN {X 0,Y 355.099,Z 237.744,A -85,B 0,C 180,E1 -13326.821,E2 -13326.821} C_VEL
LIN {X 0,Y 354.956,Z 237.741,A -85,B 0,C 180,E1 -13330.265,E2 -13330.265} C_VEL
LIN {X 0,Y 354.943,Z 237.767,A -85,B 0,C 180,E1 -13334.019,E2 -13334.019} C_VEL
LIN {X 0,Y 354.89,Z 237.752,A -85,B 0,C 180,E1 -13338.093,E2 -13338.093} C_VEL
LIN {X 0,Y 354.831,Z 237.781,A -85,B 0,C 180,E1 -13342.107,E2 -13342.107} C_VEL
LIN {X 0,Y 354.899,Z 237.762,A -85,B 0,C 180,E1 -13345.828,E2 -13345.828} C_VEL
LIN {X 0,Y 354.819,Z 237.783,A -85,B 0,C 180,E1 -13349.682,E2 -13349.682} C_VEL
LIN {X 0,Y 354.807,Z 237.772,A -85,B 0,C 180,E1 -13353.703,E2 -13353.703} C_VEL
LIN {X 0,Y 354.796,Z 237.788,A -85,B 0,C 180,E1 -13356.46,E2 -13356.46} C_VEL
LIN {X 0,Y 354.826,Z 237.776,A -85,B 0,C 180,E1 -13359.424,E2 -13359.424} C_VEL
LIN {X 0,Y 354.789,Z 237.789,A -85,B 0,C 180,E1 -13362.868,E2 -13362.868} C_VEL
LIN {X 0,Y 354.769,Z 237.794,A -85,B 0,C 180,E1 -13366.104,E2 -13366.104} C_VEL
LIN {X 0,Y 354.789,Z 237.768,A -85,B 0,C 180,E1 -13369.179,E2 -13369.179} C_VEL
LIN {X 0,Y 354.81,Z 237.789,A -85,B 0,C 180,E1 -13372.403,E2 -13372.403} C_VEL
LIN {X 0,Y 354.814,Z 237.776,A -85,B 0,C 180,E1 -13374.941,E2 -13374.941} C_VEL
LIN {X 0,Y 354.882,Z 237.987,A -85,B 0,C 180,E1 -13378.082,E2 -13378.082} C_VEL
LIN {X 0,Y 356.414,Z 245.608,A -85,B 0,C 180,E1 -13380.789,E2 -13380.789} C_VEL
LIN {X 0,Y 357.914,Z 253.975,A -85,B 0,C 180,E1 -13383.467,E2 -13383.467} C_VEL
LIN {X 0,Y 357.817,Z 257.744,A -85,B 0,C 180,E1 -13384.623,E2 -13384.623} C_VEL
LIN {X 0,Y 356.801,Z 266.878,A -85,B 0,C 180,E1 -13387.39,E2 -13387.39} C_VEL
LIN {X 0,Y 358.023,Z 272.869,A -85,B 0,C 180,E1 -13387.651,E2 -13387.651} C_VEL
LIN {X 0,Y 362.986,Z 299.416,A -85,B 0,C 180,E1 -13388.523,E2 -13388.523} C_VEL
LIN {X 0,Y 363.477,Z 302.823,A -85,B 0,C 180,E1 -13388.624,E2 -13388.624} C_VEL
LIN {X 0,Y 362.331,Z 371.714,A -85,B 0,C 180,E1 -13390.01,E2 -13390.01} C_VEL
LIN {X 0,Y 361.887,Z 381.604,A -85,B 0,C 180,E1 -13390.317,E2 -13390.317} C_VEL
LIN {X 0,Y 361.276,Z 391.579,A -85,B 0,C 180,E1 -13390.762,E2 -13390.762} C_VEL
LIN {X 0,Y 360.47,Z 401.94,A -85,B 0,C 180,E1 -13391.382,E2 -13391.382} C_VEL
LIN {X 0,Y 359.682,Z 411.074,A -85,B 0,C 180,E1 -13392.077,E2 -13392.077} C_VEL
LIN {X 0,Y 358.743,Z 420.069,A -85,B 0,C 180,E1 -13392.911,E2 -13392.911} C_VEL
LIN {X 0,Y 357.8,Z 428.797,A -85,B 0,C 180,E1 -13393.892,E2 -13393.892} C_VEL
LIN {X 0,Y 357.025,Z 436.165,A -85,B 0,C 180,E1 -13394.877,E2 -13394.877} C_VEL
LIN {X 0,Y 356.216,Z 443.414,A -85,B 0,C 180,E1 -13396.014,E2 -13396.014} C_VEL
LIN {X 0,Y 355.466,Z 449.615,A -85,B 0,C 180,E1 -13397.148,E2 -13397.148} C_VEL
LIN {X 0,Y 354.679,Z 456.151,A -85,B 0,C 180,E1 -13398.571,E2 -13398.571} C_VEL
LIN {X 0,Y 354.255,Z 460.655,A -85,B 0,C 180,E1 -13399.715,E2 -13399.715} C_VEL
LIN {X 0,Y 353.727,Z 466.146,A -85,B 0,C 180,E1 -13401.43,E2 -13401.43} C_VEL
LIN {X 0,Y 353.418,Z 470.472,A -85,B 0,C 180,E1 -13403.147,E2 -13403.147} C_VEL
LIN {X 0,Y 353.291,Z 472.839,A -85,B 0,C 180,E1 -13404.292,E2 -13404.292} C_VEL
LIN {X 0,Y 353.264,Z 474.639,A -85,B 0,C 180,E1 -13405.436,E2 -13405.436} C_VEL
LIN {X 0,Y 353.173,Z 477.084,A -85,B 0,C 180,E1 -13407.719,E2 -13407.719} C_VEL
LIN {X 0,Y 353.203,Z 477.673,A -85,B 0,C 180,E1 -13408.86,E2 -13408.86} C_VEL
LIN {X 0,Y 353.203,Z 477.673,A -85,B 0,C 180,E1 -13411.14,E2 -13411.14} C_VEL
LIN {X 0,Y 353.173,Z 477.084,A -85,B 0,C 180,E1 -13412.281,E2 -13412.281} C_VEL
LIN {X 0,Y 353.264,Z 474.639,A -85,B 0,C 180,E1 -13414.564,E2 -13414.564} C_VEL
LIN {X 0,Y 353.298,Z 472.418,A -85,B 0,C 180,E1 -13415.937,E2 -13415.937} C_VEL
LIN {X 0,Y 353.514,Z 469.232,A -85,B 0,C 180,E1 -13417.425,E2 -13417.425} C_VEL
LIN {X 0,Y 353.879,Z 464.486,A -85,B 0,C 180,E1 -13419.142,E2 -13419.142} C_VEL
LIN {X 0,Y 354.473,Z 458.464,A -85,B 0,C 180,E1 -13420.857,E2 -13420.857} C_VEL
LIN {X 0,Y 355.13,Z 452.367,A -85,B 0,C 180,E1 -13422.283,E2 -13422.283} C_VEL
LIN {X 0,Y 355.833,Z 446.667,A -85,B 0,C 180,E1 -13423.419,E2 -13423.419} C_VEL
LIN {X 0,Y 356.802,Z 438.113,A -85,B 0,C 180,E1 -13424.837,E2 -13424.837} C_VEL
LIN {X 0,Y 357.671,Z 429.932,A -85,B 0,C 180,E1 -13425.967,E2 -13425.967} C_VEL
LIN {X 0,Y 358.585,Z 421.42,A -85,B 0,C 180,E1 -13426.95,E2 -13426.95} C_VEL
LIN {X 0,Y 359.504,Z 412.706,A -85,B 0,C 180,E1 -13427.785,E2 -13427.785} C_VEL
LIN {X 0,Y 360.355,Z 402.946,A -85,B 0,C 180,E1 -13428.551,E2 -13428.551} C_VEL
LIN {X 0,Y 361.185,Z 392.866,A -85,B 0,C 180,E1 -13429.169,E2 -13429.169} C_VEL
LIN {X 0,Y 361.826,Z 383.353,A -85,B 0,C 180,E1 -13429.613,E2 -13429.613} C_VEL
LIN {X 0,Y 362.309,Z 373.04,A -85,B 0,C 180,E1 -13429.955,E2 -13429.955} C_VEL
LIN {X 0,Y 363.469,Z 302.214,A -85,B 0,C 180,E1 -13431.389,E2 -13431.389} C_VEL
LIN {X 0,Y 358.376,Z 274.544,A -85,B 0,C 180,E1 -13432.29,E2 -13432.29} C_VEL
LIN {X 0,Y 356.797,Z 267.027,A -85,B 0,C 180,E1 -13432.59,E2 -13432.59} C_VEL
LIN {X 0,Y 356.965,Z 264.811,A -85,B 0,C 180,E1 -13433.189,E2 -13433.189} C_VEL
LIN {X 0,Y 357.939,Z 257.039,A -85,B 0,C 180,E1 -13435.592,E2 -13435.592} C_VEL
LIN {X 0,Y 357.82,Z 253.038,A -85,B 0,C 180,E1 -13436.856,E2 -13436.856} C_VEL
LIN {X 0,Y 356.176,Z 244.305,A -85,B 0,C 180,E1 -13439.749,E2 -13439.749} C_VEL
LIN {X 0,Y 354.842,Z 237.803,A -85,B 0,C 180,E1 -13442.024,E2 -13442.024} C_VEL
LIN {X 0,Y 354.824,Z 237.773,A -85,B 0,C 180,E1 -13445.699,E2 -13445.699} C_VEL
LIN {X 0,Y 354.826,Z 237.768,A -85,B 0,C 180,E1 -13449.423,E2 -13449.423} C_VEL
LIN {X 0,Y 354.79,Z 237.788,A -85,B 0,C 180,E1 -13452.867,E2 -13452.867} C_VEL
LIN {X 0,Y 354.768,Z 237.789,A -85,B 0,C 180,E1 -13456.103,E2 -13456.103} C_VEL
LIN {X 0,Y 354.789,Z 237.784,A -85,B 0,C 180,E1 -13459.178,E2 -13459.178} C_VEL
LIN {X 0,Y 354.807,Z 237.787,A -85,B 0,C 180,E1 -13462.402,E2 -13462.402} C_VEL
LIN {X 0,Y 354.809,Z 237.777,A -85,B 0,C 180,E1 -13464.94,E2 -13464.94} C_VEL
LIN {X 0,Y 354.794,Z 237.787,A -85,B 0,C 180,E1 -13468.405,E2 -13468.405} C_VEL
LIN {X 0,Y 354.847,Z 237.77,A -85,B 0,C 180,E1 -13471.618,E2 -13471.618} C_VEL
LIN {X 0,Y 354.899,Z 237.762,A -85,B 0,C 180,E1 -13474.172,E2 -13474.172} C_VEL
LIN {X 0,Y 354.831,Z 237.781,A -85,B 0,C 180,E1 -13477.893,E2 -13477.893} C_VEL
LIN {X 0,Y 354.89,Z 237.752,A -85,B 0,C 180,E1 -13481.907,E2 -13481.907} C_VEL
LIN {X 0,Y 354.943,Z 237.767,A -85,B 0,C 180,E1 -13485.981,E2 -13485.981} C_VEL
LIN {X 0,Y 354.956,Z 237.741,A -85,B 0,C 180,E1 -13489.735,E2 -13489.735} C_VEL
LIN {X 0,Y 355.099,Z 237.744,A -85,B 0,C 180,E1 -13493.179,E2 -13493.179} C_VEL
LIN {X 0,Y 355.243,Z 237.723,A -85,B 0,C 180,E1 -13497.732,E2 -13497.732} C_VEL
LIN {X 0,Y 355.374,Z 237.686,A -85,B 0,C 180,E1 -13499.999,E2 -13499.999} C_VEL
LIN {X 0,Y 355.244,Z 237.718,A -85,B 0,C 180,E1 -13502.267,E2 -13502.267} C_VEL
LIN {X 0,Y 355.123,Z 237.743,A -85,B 0,C 180,E1 -13506.819,E2 -13506.819} C_VEL
LIN {X 0,Y 354.977,Z 237.737,A -85,B 0,C 180,E1 -13510.263,E2 -13510.263} C_VEL
LIN {X 0,Y 354.941,Z 237.77,A -85,B 0,C 180,E1 -13514.018,E2 -13514.018} C_VEL
LIN {X 0,Y 354.92,Z 237.753,A -85,B 0,C 180,E1 -13518.108,E2 -13518.108} C_VEL
LIN {X 0,Y 354.813,Z 237.783,A -85,B 0,C 180,E1 -13522.107,E2 -13522.107} C_VEL
LIN {X 0,Y 354.895,Z 237.766,A -85,B 0,C 180,E1 -13525.827,E2 -13525.827} C_VEL
LIN {X 0,Y 354.851,Z 237.777,A -85,B 0,C 180,E1 -13529.678,E2 -13529.678} C_VEL
LIN {X 0,Y 354.803,Z 237.777,A -85,B 0,C 180,E1 -13533.702,E2 -13533.702} C_VEL
LIN {X 0,Y 354.796,Z 237.788,A -85,B 0,C 180,E1 -13536.459,E2 -13536.459} C_VEL
LIN {X 0,Y 354.821,Z 237.783,A -85,B 0,C 180,E1 -13539.423,E2 -13539.423} C_VEL
LIN {X 0,Y 354.834,Z 237.784,A -85,B 0,C 180,E1 -13542.875,E2 -13542.875} C_VEL
LIN {X 0,Y 354.78,Z 237.768,A -85,B 0,C 180,E1 -13546.106,E2 -13546.106} C_VEL
LIN {X 0,Y 354.815,Z 237.755,A -85,B 0,C 180,E1 -13549.183,E2 -13549.183} C_VEL
LIN {X 0,Y 354.805,Z 237.788,A -85,B 0,C 180,E1 -13552.402,E2 -13552.402} C_VEL
LIN {X 0,Y 354.808,Z 237.762,A -85,B 0,C 180,E1 -13554.941,E2 -13554.941} C_VEL
LIN {X 0,Y 354.789,Z 237.791,A -85,B 0,C 180,E1 -13558.405,E2 -13558.405} C_VEL
LIN {X 0,Y 354.842,Z 237.77,A -85,B 0,C 180,E1 -13561.618,E2 -13561.618} C_VEL
LIN {X 0,Y 354.895,Z 237.78,A -85,B 0,C 180,E1 -13564.172,E2 -13564.172} C_VEL
LIN {X 0,Y 354.831,Z 237.788,A -85,B 0,C 180,E1 -13567.894,E2 -13567.894} C_VEL
LIN {X 0,Y 354.913,Z 238.03,A -85,B 0,C 180,E1 -13570.667,E2 -13570.667} C_VEL
LIN {X 0,Y 355.228,Z 239.267,A -85,B 0,C 180,E1 -13570.969,E2 -13570.969} C_VEL
LIN {X 0,Y 356.951,Z 241.981,A -85,B 0,C 180,E1 -13571.466,E2 -13571.466} C_VEL
LIN {X 0,Y 359.163,Z 243.77,A -85,B 0,C 180,E1 -13572.034,E2 -13572.034} C_VEL
LIN {X 0,Y 361.199,Z 246.944,A -85,B 0,C 180,E1 -13572.646,E2 -13572.646} C_VEL
LIN {X 0,Y 363.774,Z 248.964,A -85,B 0,C 180,E1 -13573.342,E2 -13573.342} C_VEL
LIN {X 0,Y 366.387,Z 252.552,A -85,B 0,C 180,E1 -13574.187,E2 -13574.187} C_VEL
LIN {X 0,Y 369.304,Z 254.875,A -85,B 0,C 180,E1 -13575.084,E2 -13575.084} C_VEL
LIN {X 0,Y 372.95,Z 259.199,A -85,B 0,C 180,E1 -13576.358,E2 -13576.358} C_VEL
LIN {X 0,Y 376.191,Z 261.732,A -85,B 0,C 180,E1 -13577.559,E2 -13577.559} C_VEL
LIN {X 0,Y 379.015,Z 265.137,A -85,B 0,C 180,E1 -13578.786,E2 -13578.786} C_VEL
LIN {X 0,Y 381.764,Z 267.214,A -85,B 0,C 180,E1 -13580.044,E2 -13580.044} C_VEL
LIN {X 0,Y 383.693,Z 268.296,A -85,B 0,C 180,E1 -13580.976,E2 -13580.976} C_VEL
LIN {X 0,Y 386.239,Z 271.58,A -85,B 0,C 180,E1 -13582.578,E2 -13582.578} C_VEL
LIN {X 0,Y 388.478,Z 273.435,A -85,B 0,C 180,E1 -13584.267,E2 -13584.267} C_VEL
LIN {X 0,Y 390.135,Z 274.324,A -85,B 0,C 180,E1 -13585.868,E2 -13585.868} C_VEL
LIN {X 0,Y 391.262,Z 274.7,A -85,B 0,C 180,E1 -13587.445,E2 -13587.445} C_VEL
LIN {X 0,Y 391.823,Z 275.132,A -85,B 0,C 180,E1 -13588.972,E2 -13588.972} C_VEL
LIN {X 0,Y 391.999,Z 275.069,A -85,B 0,C 180,E1 -13590,E2 -13590} C_VEL
LIN {X 0,Y 391.73,Z 275.018,A -85,B 0,C 180,E1 -13591.542,E2 -13591.542} C_VEL
LIN {X 0,Y 390.988,Z 274.588,A -85,B 0,C 180,E1 -13593.091,E2 -13593.091} C_VEL
LIN {X 0,Y 389.394,Z 273.976,A -85,B 0,C 180,E1 -13594.918,E2 -13594.918} C_VEL
LIN {X 0,Y 387.3,Z 272.542,A -85,B 0,C 180,E1 -13596.652,E2 -13596.652} C_VEL
LIN {X 0,Y 385.253,Z 270.468,A -85,B 0,C 180,E1 -13598.052,E2 -13598.052} C_VEL
LIN {X 0,Y 383.438,Z 268.005,A -85,B 0,C 180,E1 -13599.167,E2 -13599.167} C_VEL
LIN {X 0,Y 380.179,Z 266.112,A -85,B 0,C 180,E1 -13600.72,E2 -13600.72} C_VEL
LIN {X 0,Y 377.084,Z 262.937,A -85,B 0,C 180,E1 -13602.069,E2 -13602.069} C_VEL
LIN {X 0,Y 375.687,Z 261.212,A -85,B 0,C 180,E1 -13602.629,E2 -13602.629} C_VEL
LIN {X 0,Y 372.563,Z 258.795,A -85,B 0,C 180,E1 -13603.784,E2 -13603.784} C_VEL
LIN {X 0,Y 369.831,Z 255.395,A -85,B 0,C 180,E1 -13604.735,E2 -13604.735} C_VEL
LIN {X 0,Y 366.123,Z 252.303,A -85,B 0,C 180,E1 -13605.893,E2 -13605.893} C_VEL
LIN {X 0,Y 363.644,Z 248.903,A -85,B 0,C 180,E1 -13606.693,E2 -13606.693} C_VEL
LIN {X 0,Y 360.934,Z 246.667,A -85,B 0,C 180,E1 -13607.427,E2 -13607.427} C_VEL
LIN {X 0,Y 358.716,Z 243.21,A -85,B 0,C 180,E1 -13608.097,E2 -13608.097} C_VEL
LIN {X 0,Y 356.497,Z 241.476,A -85,B 0,C 180,E1 -13608.649,E2 -13608.649} C_VEL
LIN {X 0,Y 355.028,Z 238.604,A -85,B 0,C 180,E1 -13609.14,E2 -13609.14} C_VEL
LIN {X 0,Y 354.861,Z 237.836,A -85,B 0,C 180,E1 -13609.524,E2 -13609.524} C_VEL
LIN {X 0,Y 354.828,Z 237.788,A -85,B 0,C 180,E1 -13613.337,E2 -13613.337} C_VEL
LIN {X 0,Y 354.884,Z 237.781,A -85,B 0,C 180,E1 -13616.982,E2 -13616.982} C_VEL
LIN {X 0,Y 354.814,Z 237.767,A -85,B 0,C 180,E1 -13619.682,E2 -13619.682} C_VEL
LIN {X 0,Y 354.81,Z 237.767,A -85,B 0,C 180,E1 -13623.684,E2 -13623.684} C_VEL
LIN {X 0,Y 354.795,Z 237.779,A -85,B 0,C 180,E1 -13626.46,E2 -13626.46} C_VEL
LIN {X 0,Y 354.82,Z 237.779,A -85,B 0,C 180,E1 -13629.424,E2 -13629.424} C_VEL
LIN {X 0,Y 354.789,Z 237.753,A -85,B 0,C 180,E1 -13632.868,E2 -13632.868} C_VEL
LIN {X 0,Y 354.849,Z 237.784,A -85,B 0,C 180,E1 -13636.117,E2 -13636.117} C_VEL
LIN {X 0,Y 354.823,Z 237.773,A -85,B 0,C 180,E1 -13639.588,E2 -13639.588} C_VEL
LIN {X 0,Y 354.797,Z 237.788,A -85,B 0,C 180,E1 -13643.541,E2 -13643.541} C_VEL
LIN {X 0,Y 354.811,Z 237.775,A -85,B 0,C 180,E1 -13644.523,E2 -13644.523} C_VEL
LIN {X 0,Y 354.12,Z 237.86,A -85,B 0,C 180,E1 -13645.47,E2 -13645.47} C_VEL
LIN {X 0,Y 351.225,Z 238.227,A -85,B 0,C 180,E1 -13647.009,E2 -13647.009} C_VEL
LIN {X 0,Y 348.809,Z 238.537,A -85,B 0,C 180,E1 -13648.255,E2 -13648.255} C_VEL
LIN {X 0,Y 347.812,Z 238.66,A -85,B 0,C 180,E1 -13649.22,E2 -13649.22} C_VEL
LIN {X 0,Y 347.752,Z 238.668,A -85,B 0,C 180,E1 -13649.546,E2 -13649.546} C_VEL
LIN {X 0,Y 347.848,Z 238.63,A -85,B 0,C 180,E1 -13652.746,E2 -13652.746} C_VEL
LIN {X 0,Y 347.782,Z 238.664,A -85,B 0,C 180,E1 -13656.162,E2 -13656.162} C_VEL
LIN {X 0,Y 347.804,Z 238.637,A -85,B 0,C 180,E1 -13659.91,E2 -13659.91} C_VEL
LIN {X 0,Y 347.864,Z 238.639,A -85,B 0,C 180,E1 -13662.36,E2 -13662.36} C_VEL
LIN {X 0,Y 347.896,Z 238.647,A -85,B 0,C 180,E1 -13665.971,E2 -13665.971} C_VEL
LIN {X 0,Y 347.927,Z 238.615,A -85,B 0,C 180,E1 -13669.526,E2 -13669.526} C_VEL
LIN {X 0,Y 348.089,Z 238.617,A -85,B 0,C 180,E1 -13673.043,E2 -13673.043} C_VEL
LIN {X 0,Y 348.207,Z 238.594,A -85,B 0,C 180,E1 -13677.687,E2 -13677.687} C_VEL
LIN {X 0,Y 348.324,Z 238.563,A -85,B 0,C 180,E1 -13680.001,E2 -13680.001} C_VEL
LIN {X 0,Y 348.206,Z 238.6,A -85,B 0,C 180,E1 -13682.314,E2 -13682.314} C_VEL
LIN {X 0,Y 348.067,Z 238.618,A -85,B 0,C 180,E1 -13686.959,E2 -13686.959} C_VEL
LIN {X 0,Y 347.896,Z 238.621,A -85,B 0,C 180,E1 -13690.476,E2 -13690.476} C_VEL
LIN {X 0,Y 347.899,Z 238.645,A -85,B 0,C 180,E1 -13694.15,E2 -13694.15} C_VEL
LIN {X 0,Y 347.829,Z 238.63,A -85,B 0,C 180,E1 -13698.26,E2 -13698.26} C_VEL
LIN {X 0,Y 347.787,Z 238.657,A -85,B 0,C 180,E1 -13701.635,E2 -13701.635} C_VEL
LIN {X 0,Y 347.812,Z 238.647,A -85,B 0,C 180,E1 -13705.109,E2 -13705.109} C_VEL
LIN {X 0,Y 347.809,Z 238.642,A -85,B 0,C 180,E1 -13707.695,E2 -13707.695} C_VEL
LIN {X 0,Y 347.75,Z 238.668,A -85,B 0,C 180,E1 -13710.348,E2 -13710.348} C_VEL
LIN {X 0,Y 347.749,Z 238.65,A -85,B 0,C 180,E1 -13714.044,E2 -13714.044} C_VEL
LIN {X 0,Y 347.761,Z 238.665,A -85,B 0,C 180,E1 -13717.322,E2 -13717.322} C_VEL
LIN {X 0,Y 347.733,Z 238.659,A -85,B 0,C 180,E1 -13720.298,E2 -13720.298} C_VEL
LIN {X 0,Y 347.725,Z 238.668,A -85,B 0,C 180,E1 -13723.409,E2 -13723.409} C_VEL
LIN {X 0,Y 347.727,Z 238.671,A -85,B 0,C 180,E1 -13726.687,E2 -13726.687} C_VEL
LIN {X 0,Y 347.749,Z 238.645,A -85,B 0,C 180,E1 -13730.174,E2 -13730.174} C_VEL
LIN {X 0,Y 347.764,Z 238.665,A -85,B 0,C 180,E1 -13732.68,E2 -13732.68} C_VEL
LIN {X 0,Y 347.751,Z 238.668,A -85,B 0,C 180,E1 -13735.957,E2 -13735.957} C_VEL
LIN {X 0,Y 347.819,Z 238.839,A -85,B 0,C 180,E1 -13737.704,E2 -13737.704} C_VEL
LIN {X 0,Y 349.433,Z 246.756,A -85,B 0,C 180,E1 -13740.569,E2 -13740.569} C_VEL
LIN {X 0,Y 350.918,Z 254.839,A -85,B 0,C 180,E1 -13743.217,E2 -13743.217} C_VEL
LIN {X 0,Y 350.917,Z 258.272,A -85,B 0,C 180,E1 -13744.322,E2 -13744.322} C_VEL
LIN {X 0,Y 349.943,Z 266.62,A -85,B 0,C 180,E1 -13746.91,E2 -13746.91} C_VEL
LIN {X 0,Y 350.634,Z 270.349,A -85,B 0,C 180,E1 -13747.104,E2 -13747.104} C_VEL
LIN {X 0,Y 355.43,Z 294.558,A -85,B 0,C 180,E1 -13747.944,E2 -13747.944} C_VEL
LIN {X 0,Y 356.836,Z 304.088,A -85,B 0,C 180,E1 -13748.237,E2 -13748.237} C_VEL
LIN {X 0,Y 355.689,Z 371.529,A -85,B 0,C 180,E1 -13749.62,E2 -13749.62} C_VEL
LIN {X 0,Y 355.212,Z 381.411,A -85,B 0,C 180,E1 -13749.931,E2 -13749.931} C_VEL
LIN {X 0,Y 354.585,Z 391.386,A -85,B 0,C 180,E1 -13750.385,E2 -13750.385} C_VEL
LIN {X 0,Y 353.761,Z 401.748,A -85,B 0,C 180,E1 -13751.016,E2 -13751.016} C_VEL
LIN {X 0,Y 352.905,Z 410.881,A -85,B 0,C 180,E1 -13751.72,E2 -13751.72} C_VEL
LIN {X 0,Y 351.969,Z 419.877,A -85,B 0,C 180,E1 -13752.572,E2 -13752.572} C_VEL
LIN {X 0,Y 350.949,Z 428.603,A -85,B 0,C 180,E1 -13753.569,E2 -13753.569} C_VEL
LIN {X 0,Y 350.072,Z 436.684,A -85,B 0,C 180,E1 -13754.68,E2 -13754.68} C_VEL
LIN {X 0,Y 349.076,Z 444.846,A -85,B 0,C 180,E1 -13756.019,E2 -13756.019} C_VEL
LIN {X 0,Y 348.336,Z 450.797,A -85,B 0,C 180,E1 -13757.177,E2 -13757.177} C_VEL
LIN {X 0,Y 347.56,Z 457.113,A -85,B 0,C 180,E1 -13758.629,E2 -13758.629} C_VEL
LIN {X 0,Y 347.019,Z 462.377,A -85,B 0,C 180,E1 -13760.087,E2 -13760.087} C_VEL
LIN {X 0,Y 346.552,Z 467.507,A -85,B 0,C 180,E1 -13761.839,E2 -13761.839} C_VEL
LIN {X 0,Y 346.284,Z 471.497,A -85,B 0,C 180,E1 -13763.592,E2 -13763.592} C_VEL
LIN {X 0,Y 346.162,Z 474.446,A -85,B 0,C 180,E1 -13765.342,E2 -13765.342} C_VEL
LIN {X 0,Y 346.084,Z 476.891,A -85,B 0,C 180,E1 -13767.672,E2 -13767.672} C_VEL
LIN {X 0,Y 346.104,Z 477.481,A -85,B 0,C 180,E1 -13768.836,E2 -13768.836} C_VEL
LIN {X 0,Y 346.104,Z 477.481,A -85,B 0,C 180,E1 -13771.164,E2 -13771.164} C_VEL
LIN {X 0,Y 346.084,Z 476.891,A -85,B 0,C 180,E1 -13772.328,E2 -13772.328} C_VEL
LIN {X 0,Y 346.161,Z 474.446,A -85,B 0,C 180,E1 -13774.658,E2 -13774.658} C_VEL
LIN {X 0,Y 346.247,Z 471.496,A -85,B 0,C 180,E1 -13776.409,E2 -13776.409} C_VEL
LIN {X 0,Y 346.552,Z 467.507,A -85,B 0,C 180,E1 -13778.161,E2 -13778.161} C_VEL
LIN {X 0,Y 347.019,Z 462.377,A -85,B 0,C 180,E1 -13779.913,E2 -13779.913} C_VEL
LIN {X 0,Y 347.56,Z 457.113,A -85,B 0,C 180,E1 -13781.371,E2 -13781.371} C_VEL
LIN {X 0,Y 348.333,Z 450.797,A -85,B 0,C 180,E1 -13782.823,E2 -13782.823} C_VEL
LIN {X 0,Y 349.057,Z 444.846,A -85,B 0,C 180,E1 -13783.982,E2 -13783.982} C_VEL
LIN {X 0,Y 350.042,Z 436.808,A -85,B 0,C 180,E1 -13785.302,E2 -13785.302} C_VEL
LIN {X 0,Y 350.949,Z 428.603,A -85,B 0,C 180,E1 -13786.431,E2 -13786.431} C_VEL
LIN {X 0,Y 351.955,Z 419.876,A -85,B 0,C 180,E1 -13787.429,E2 -13787.429} C_VEL
LIN {X 0,Y 352.907,Z 410.881,A -85,B 0,C 180,E1 -13788.28,E2 -13788.28} C_VEL
LIN {X 0,Y 353.847,Z 400.741,A -85,B 0,C 180,E1 -13789.055,E2 -13789.055} C_VEL
LIN {X 0,Y 354.804,Z 388.812,A -85,B 0,C 180,E1 -13789.754,E2 -13789.754} C_VEL
LIN {X 0,Y 355.571,Z 375.512,A -85,B 0,C 180,E1 -13790.274,E2 -13790.274} C_VEL
LIN {X 0,Y 356.049,Z 356.729,A -85,B 0,C 180,E1 -13790.698,E2 -13790.698} C_VEL
LIN {X 0,Y 356.829,Z 302.937,A -85,B 0,C 180,E1 -13791.788,E2 -13791.788} C_VEL
LIN {X 0,Y 352.182,Z 277.435,A -85,B 0,C 180,E1 -13792.637,E2 -13792.637} C_VEL
LIN {X 0,Y 349.939,Z 266.901,A -85,B 0,C 180,E1 -13793.051,E2 -13793.051} C_VEL
LIN {X 0,Y 350,Z 265.561,A -85,B 0,C 180,E1 -13793.365,E2 -13793.365} C_VEL
LIN {X 0,Y 351.042,Z 256.844,A -85,B 0,C 180,E1 -13796.132,E2 -13796.132} C_VEL
LIN {X 0,Y 350.316,Z 251.138,A -85,B 0,C 180,E1 -13798.026,E2 -13798.026} C_VEL
LIN {X 0,Y 348.209,Z 240.585,A -85,B 0,C 180,E1 -13801.652,E2 -13801.652} C_VEL
LIN {X 0,Y 347.793,Z 238.706,A -85,B 0,C 180,E1 -13802.375,E2 -13802.375} C_VEL
LIN {X 0,Y 347.772,Z 238.652,A -85,B 0,C 180,E1 -13806.065,E2 -13806.065} C_VEL
LIN {X 0,Y 347.754,Z 238.66,A -85,B 0,C 180,E1 -13808.792,E2 -13808.792} C_VEL
LIN {X 0,Y 347.752,Z 238.653,A -85,B 0,C 180,E1 -13811.83,E2 -13811.83} C_VEL
LIN {X 0,Y 347.707,Z 238.667,A -85,B 0,C 180,E1 -13815.026,E2 -13815.026} C_VEL
LIN {X 0,Y 347.752,Z 238.664,A -85,B 0,C 180,E1 -13818.397,E2 -13818.397} C_VEL
LIN {X 0,Y 347.773,Z 238.665,A -85,B 0,C 180,E1 -13822.011,E2 -13822.011} C_VEL
LIN {X 0,Y 347.743,Z 238.651,A -85,B 0,C 180,E1 -13825.535,E2 -13825.535} C_VEL
LIN {X 0,Y 347.745,Z 238.665,A -85,B 0,C 180,E1 -13828.3,E2 -13828.3} C_VEL
LIN {X 0,Y 347.78,Z 238.658,A -85,B 0,C 180,E1 -13830.987,E2 -13830.987} C_VEL
LIN {X 0,Y 347.831,Z 238.636,A -85,B 0,C 180,E1 -13833.607,E2 -13833.607} C_VEL
LIN {X 0,Y 347.786,Z 238.659,A -85,B 0,C 180,E1 -13836.161,E2 -13836.161} C_VEL
LIN {X 0,Y 347.803,Z 238.642,A -85,B 0,C 180,E1 -13839.908,E2 -13839.908} C_VEL
LIN {X 0,Y 347.832,Z 238.647,A -85,B 0,C 180,E1 -13843.568,E2 -13843.568} C_VEL
LIN {X 0,Y 347.89,Z 238.644,A -85,B 0,C 180,E1 -13847.16,E2 -13847.16} C_VEL
LIN {X 0,Y 347.935,Z 238.612,A -85,B 0,C 180,E1 -13850.7,E2 -13850.7} C_VEL
LIN {X 0,Y 348.067,Z 238.618,A -85,B 0,C 180,E1 -13853.041,E2 -13853.041} C_VEL
LIN {X 0,Y 348.206,Z 238.6,A -85,B 0,C 180,E1 -13857.686,E2 -13857.686} C_VEL
LIN {X 0,Y 348.324,Z 238.563,A -85,B 0,C 180,E1 -13859.999,E2 -13859.999} C_VEL
LIN {X 0,Y 348.207,Z 238.594,A -85,B 0,C 180,E1 -13862.313,E2 -13862.313} C_VEL
LIN {X 0,Y 348.089,Z 238.617,A -85,B 0,C 180,E1 -13866.957,E2 -13866.957} C_VEL
LIN {X 0,Y 347.927,Z 238.615,A -85,B 0,C 180,E1 -13870.474,E2 -13870.474} C_VEL
LIN {X 0,Y 347.897,Z 238.648,A -85,B 0,C 180,E1 -13874.149,E2 -13874.149} C_VEL
LIN {X 0,Y 347.889,Z 238.626,A -85,B 0,C 180,E1 -13878.289,E2 -13878.289} C_VEL
LIN {X 0,Y 347.765,Z 238.658,A -85,B 0,C 180,E1 -13881.626,E2 -13881.626} C_VEL
LIN {X 0,Y 347.809,Z 238.653,A -85,B 0,C 180,E1 -13885.108,E2 -13885.108} C_VEL
LIN {X 0,Y 347.807,Z 238.636,A -85,B 0,C 180,E1 -13887.693,E2 -13887.693} C_VEL
LIN {X 0,Y 347.761,Z 238.667,A -85,B 0,C 180,E1 -13890.346,E2 -13890.346} C_VEL
LIN {X 0,Y 347.741,Z 238.652,A -85,B 0,C 180,E1 -13894.463,E2 -13894.463} C_VEL
LIN {X 0,Y 347.772,Z 238.669,A -85,B 0,C 180,E1 -13897.989,E2 -13897.989} C_VEL
LIN {X 0,Y 347.782,Z 238.653,A -85,B 0,C 180,E1 -13901.609,E2 -13901.609} C_VEL
LIN {X 0,Y 347.793,Z 238.656,A -85,B 0,C 180,E1 -13905.011,E2 -13905.011} C_VEL
LIN {X 0,Y 347.758,Z 238.624,A -85,B 0,C 180,E1 -13908.395,E2 -13908.395} C_VEL
LIN {X 0,Y 347.772,Z 238.667,A -85,B 0,C 180,E1 -13912.01,E2 -13912.01} C_VEL
LIN {X 0,Y 347.74,Z 238.641,A -85,B 0,C 180,E1 -13915.536,E2 -13915.536} C_VEL
LIN {X 0,Y 347.741,Z 238.67,A -85,B 0,C 180,E1 -13918.3,E2 -13918.3} C_VEL
LIN {X 0,Y 347.774,Z 238.644,A -85,B 0,C 180,E1 -13920.987,E2 -13920.987} C_VEL
LIN {X 0,Y 347.827,Z 238.661,A -85,B 0,C 180,E1 -13923.608,E2 -13923.608} C_VEL
LIN {X 0,Y 347.785,Z 238.666,A -85,B 0,C 180,E1 -13926.162,E2 -13926.162} C_VEL
LIN {X 0,Y 347.821,Z 238.782,A -85,B 0,C 180,E1 -13929.138,E2 -13929.138} C_VEL
LIN {X 0,Y 348.019,Z 239.797,A -85,B 0,C 180,E1 -13929.459,E2 -13929.459} C_VEL
LIN {X 0,Y 349.6,Z 242.552,A -85,B 0,C 180,E1 -13929.906,E2 -13929.906} C_VEL
LIN {X 0,Y 351.803,Z 244.458,A -85,B 0,C 180,E1 -13930.408,E2 -13930.408} C_VEL
LIN {X 0,Y 353.932,Z 247.741,A -85,B 0,C 180,E1 -13930.994,E2 -13930.994} C_VEL
LIN {X 0,Y 356.535,Z 250.131,A -85,B 0,C 180,E1 -13931.644,E2 -13931.644} C_VEL
LIN {X 0,Y 359.05,Z 253.498,A -85,B 0,C 180,E1 -13932.356,E2 -13932.356} C_VEL
LIN {X 0,Y 361.878,Z 256.009,A -85,B 0,C 180,E1 -13933.126,E2 -13933.126} C_VEL
LIN {X 0,Y 364.51,Z 259.261,A -85,B 0,C 180,E1 -13933.938,E2 -13933.938} C_VEL
LIN {X 0,Y 367.946,Z 262.102,A -85,B 0,C 180,E1 -13934.974,E2 -13934.974} C_VEL
LIN {X 0,Y 371.141,Z 265.826,A -85,B 0,C 180,E1 -13936.082,E2 -13936.082} C_VEL
LIN {X 0,Y 374.573,Z 268.556,A -85,B 0,C 180,E1 -13937.329,E2 -13937.329} C_VEL
LIN {X 0,Y 377.469,Z 271.846,A -85,B 0,C 180,E1 -13938.533,E2 -13938.533} C_VEL
LIN {X 0,Y 380.375,Z 274.048,A -85,B 0,C 180,E1 -13939.816,E2 -13939.816} C_VEL
LIN {X 0,Y 382.425,Z 275.251,A -85,B 0,C 180,E1 -13940.794,E2 -13940.794} C_VEL
LIN {X 0,Y 385.153,Z 278.56,A -85,B 0,C 180,E1 -13942.452,E2 -13942.452} C_VEL
LIN {X 0,Y 387.586,Z 280.491,A -85,B 0,C 180,E1 -13944.254,E2 -13944.254} C_VEL
LIN {X 0,Y 389.26,Z 281.369,A -85,B 0,C 180,E1 -13945.859,E2 -13945.859} C_VEL
LIN {X 0,Y 390.395,Z 281.749,A -85,B 0,C 180,E1 -13947.439,E2 -13947.439} C_VEL
LIN {X 0,Y 390.961,Z 282.178,A -85,B 0,C 180,E1 -13948.97,E2 -13948.97} C_VEL
LIN {X 0,Y 391.134,Z 282.115,A -85,B 0,C 180,E1 -13950,E2 -13950} C_VEL
LIN {X 0,Y 390.864,Z 282.038,A -85,B 0,C 180,E1 -13951.546,E2 -13951.546} C_VEL
LIN {X 0,Y 390.115,Z 281.607,A -85,B 0,C 180,E1 -13953.098,E2 -13953.098} C_VEL
LIN {X 0,Y 388.503,Z 281.029,A -85,B 0,C 180,E1 -13954.929,E2 -13954.929} C_VEL
LIN {X 0,Y 386.383,Z 279.647,A -85,B 0,C 180,E1 -13956.668,E2 -13956.668} C_VEL
LIN {X 0,Y 384.174,Z 277.561,A -85,B 0,C 180,E1 -13958.143,E2 -13958.143} C_VEL
LIN {X 0,Y 382.054,Z 274.874,A -85,B 0,C 180,E1 -13959.396,E2 -13959.396} C_VEL
LIN {X 0,Y 378.834,Z 272.988,A -85,B 0,C 180,E1 -13960.894,E2 -13960.894} C_VEL
LIN {X 0,Y 375.551,Z 269.776,A -85,B 0,C 180,E1 -13962.291,E2 -13962.291} C_VEL
LIN {X 0,Y 373.856,Z 267.855,A -85,B 0,C 180,E1 -13962.942,E2 -13962.942} C_VEL
LIN {X 0,Y 370.642,Z 265.351,A -85,B 0,C 180,E1 -13964.084,E2 -13964.084} C_VEL
LIN {X 0,Y 367.17,Z 261.329,A -85,B 0,C 180,E1 -13965.274,E2 -13965.274} C_VEL
LIN {X 0,Y 363.714,Z 258.423,A -85,B 0,C 180,E1 -13966.311,E2 -13966.311} C_VEL
LIN {X 0,Y 360.955,Z 255.102,A -85,B 0,C 180,E1 -13967.125,E2 -13967.125} C_VEL
LIN {X 0,Y 358.034,Z 252.332,A -85,B 0,C 180,E1 -13967.937,E2 -13967.937} C_VEL
LIN {X 0,Y 356.111,Z 249.541,A -85,B 0,C 180,E1 -13968.467,E2 -13968.467} C_VEL
LIN {X 0,Y 353.385,Z 247.088,A -85,B 0,C 180,E1 -13969.15,E2 -13969.15} C_VEL
LIN {X 0,Y 351.282,Z 243.921,A -85,B 0,C 180,E1 -13969.718,E2 -13969.718} C_VEL
LIN {X 0,Y 349.024,Z 241.879,A -85,B 0,C 180,E1 -13970.231,E2 -13970.231} C_VEL
LIN {X 0,Y 347.918,Z 239.335,A -85,B 0,C 180,E1 -13970.624,E2 -13970.624} C_VEL
LIN {X 0,Y 347.812,Z 238.699,A -85,B 0,C 180,E1 -13971.018,E2 -13971.018} C_VEL
LIN {X 0,Y 347.808,Z 238.662,A -85,B 0,C 180,E1 -13975.109,E2 -13975.109} C_VEL
LIN {X 0,Y 347.804,Z 238.657,A -85,B 0,C 180,E1 -13977.694,E2 -13977.694} C_VEL
LIN {X 0,Y 347.745,Z 238.653,A -85,B 0,C 180,E1 -13980.348,E2 -13980.348} C_VEL
LIN {X 0,Y 347.744,Z 238.643,A -85,B 0,C 180,E1 -13984.044,E2 -13984.044} C_VEL
LIN {X 0,Y 347.759,Z 238.665,A -85,B 0,C 180,E1 -13987.321,E2 -13987.321} C_VEL
LIN {X 0,Y 347.748,Z 238.644,A -85,B 0,C 180,E1 -13990.295,E2 -13990.295} C_VEL
LIN {X 0,Y 347.726,Z 238.639,A -85,B 0,C 180,E1 -13993.407,E2 -13993.407} C_VEL
LIN {X 0,Y 347.811,Z 238.66,A -85,B 0,C 180,E1 -13996.671,E2 -13996.671} C_VEL
LIN {X 0,Y 347.783,Z 238.653,A -85,B 0,C 180,E1 -14000.166,E2 -14000.166} C_VEL
LIN {X 0,Y 347.786,Z 238.653,A -85,B 0,C 180,E1 -14004.125,E2 -14004.125} C_VEL
LIN {X 0,Y 347.736,Z 238.671,A -85,B 0,C 180,E1 -14008.086,E2 -14008.086} C_VEL
LIN {X 0,Y 347.752,Z 238.668,A -85,B 0,C 180,E1 -14009.546,E2 -14009.546} C_VEL
LIN {X 0,Y 347.145,Z 238.747,A -85,B 0,C 180,E1 -14010.514,E2 -14010.514} C_VEL
LIN {X 0,Y 344.322,Z 239.094,A -85,B 0,C 180,E1 -14012.089,E2 -14012.089} C_VEL
LIN {X 0,Y 341.893,Z 239.39,A -85,B 0,C 180,E1 -14013.364,E2 -14013.364} C_VEL
LIN {X 0,Y 340.844,Z 239.519,A -85,B 0,C 180,E1 -14014.35,E2 -14014.35} C_VEL
LIN {X 0,Y 340.758,Z 239.53,A -85,B 0,C 180,E1 -14014.684,E2 -14014.684} C_VEL
LIN {X 0,Y 340.739,Z 239.534,A -85,B 0,C 180,E1 -14018.207,E2 -14018.207} C_VEL
LIN {X 0,Y 340.856,Z 239.505,A -85,B 0,C 180,E1 -14021.985,E2 -14021.985} C_VEL
LIN {X 0,Y 340.868,Z 239.525,A -85,B 0,C 180,E1 -14025.706,E2 -14025.706} C_VEL
LIN {X 0,Y 340.87,Z 239.495,A -85,B 0,C 180,E1 -14029.307,E2 -14029.307} C_VEL
LIN {X 0,Y 341.057,Z 239.492,A -85,B 0,C 180,E1 -14032.899,E2 -14032.899} C_VEL
LIN {X 0,Y 341.168,Z 239.471,A -85,B 0,C 180,E1 -14037.639,E2 -14037.639} C_VEL
LIN {X 0,Y 341.275,Z 239.441,A -85,B 0,C 180,E1 -14040.001,E2 -14040.001} C_VEL
LIN {X 0,Y 341.167,Z 239.477,A -85,B 0,C 180,E1 -14042.362,E2 -14042.362} C_VEL
LIN {X 0,Y 341.016,Z 239.494,A -85,B 0,C 180,E1 -14047.104,E2 -14047.104} C_VEL
LIN {X 0,Y 340.848,Z 239.499,A -85,B 0,C 180,E1 -14050.695,E2 -14050.695} C_VEL
LIN {X 0,Y 340.863,Z 239.522,A -85,B 0,C 180,E1 -14054.325,E2 -14054.325} C_VEL
LIN {X 0,Y 340.786,Z 239.506,A -85,B 0,C 180,E1 -14058.441,E2 -14058.441} C_VEL
LIN {X 0,Y 340.754,Z 239.533,A -85,B 0,C 180,E1 -14061.857,E2 -14061.857} C_VEL
LIN {X 0,Y 340.772,Z 239.521,A -85,B 0,C 180,E1 -14065.665,E2 -14065.665} C_VEL
LIN {X 0,Y 340.729,Z 239.527,A -85,B 0,C 180,E1 -14068.321,E2 -14068.321} C_VEL
LIN {X 0,Y 340.698,Z 239.545,A -85,B 0,C 180,E1 -14071.045,E2 -14071.045} C_VEL
LIN {X 0,Y 340.717,Z 239.534,A -85,B 0,C 180,E1 -14075.28,E2 -14075.28} C_VEL
LIN {X 0,Y 340.71,Z 239.541,A -85,B 0,C 180,E1 -14078.386,E2 -14078.386} C_VEL
LIN {X 0,Y 340.7,Z 239.545,A -85,B 0,C 180,E1 -14082.046,E2 -14082.046} C_VEL
LIN {X 0,Y 340.654,Z 239.554,A -85,B 0,C 180,E1 -14086.227,E2 -14086.227} C_VEL
LIN {X 0,Y 340.689,Z 239.522,A -85,B 0,C 180,E1 -14089.754,E2 -14089.754} C_VEL
LIN {X 0,Y 340.707,Z 239.537,A -85,B 0,C 180,E1 -14093.259,E2 -14093.259} C_VEL
LIN {X 0,Y 340.728,Z 239.543,A -85,B 0,C 180,E1 -14097.13,E2 -14097.13} C_VEL
LIN {X 0,Y 340.973,Z 240.631,A -85,B 0,C 180,E1 -14097.681,E2 -14097.681} C_VEL
LIN {X 0,Y 342.537,Z 248.377,A -85,B 0,C 180,E1 -14100.5,E2 -14100.5} C_VEL
LIN {X 0,Y 344.027,Z 256.645,A -85,B 0,C 180,E1 -14103.293,E2 -14103.293} C_VEL
LIN {X 0,Y 343.796,Z 260.57,A -85,B 0,C 180,E1 -14104.578,E2 -14104.578} C_VEL
LIN {X 0,Y 343.068,Z 266.359,A -85,B 0,C 180,E1 -14106.407,E2 -14106.407} C_VEL
LIN {X 0,Y 343.395,Z 268.47,A -85,B 0,C 180,E1 -14106.556,E2 -14106.556} C_VEL
LIN {X 0,Y 348.369,Z 292.834,A -85,B 0,C 180,E1 -14107.44,E2 -14107.44} C_VEL
LIN {X 0,Y 350.239,Z 304.97,A -85,B 0,C 180,E1 -14107.829,E2 -14107.829} C_VEL
LIN {X 0,Y 349.054,Z 371.343,A -85,B 0,C 180,E1 -14109.215,E2 -14109.215} C_VEL
LIN {X 0,Y 348.555,Z 381.218,A -85,B 0,C 180,E1 -14109.531,E2 -14109.531} C_VEL
LIN {X 0,Y 347.912,Z 391.193,A -85,B 0,C 180,E1 -14109.992,E2 -14109.992} C_VEL
LIN {X 0,Y 347.037,Z 401.555,A -85,B 0,C 180,E1 -14110.633,E2 -14110.633} C_VEL
LIN {X 0,Y 346.164,Z 410.688,A -85,B 0,C 180,E1 -14111.351,E2 -14111.351} C_VEL
LIN {X 0,Y 345.194,Z 419.684,A -85,B 0,C 180,E1 -14112.218,E2 -14112.218} C_VEL
LIN {X 0,Y 344.115,Z 428.41,A -85,B 0,C 180,E1 -14113.233,E2 -14113.233} C_VEL
LIN {X 0,Y 343.185,Z 436.611,A -85,B 0,C 180,E1 -14114.383,E2 -14114.383} C_VEL
LIN {X 0,Y 342.15,Z 444.652,A -85,B 0,C 180,E1 -14115.73,E2 -14115.73} C_VEL
LIN {X 0,Y 341.388,Z 450.604,A -85,B 0,C 180,E1 -14116.912,E2 -14116.912} C_VEL
LIN {X 0,Y 340.566,Z 456.92,A -85,B 0,C 180,E1 -14118.393,E2 -14118.393} C_VEL
LIN {X 0,Y 339.996,Z 462.183,A -85,B 0,C 180,E1 -14119.881,E2 -14119.881} C_VEL
LIN {X 0,Y 339.512,Z 467.314,A -85,B 0,C 180,E1 -14121.668,E2 -14121.668} C_VEL
LIN {X 0,Y 339.205,Z 471.303,A -85,B 0,C 180,E1 -14123.457,E2 -14123.457} C_VEL
LIN {X 0,Y 339.064,Z 474.252,A -85,B 0,C 180,E1 -14125.244,E2 -14125.244} C_VEL
LIN {X 0,Y 338.999,Z 476.699,A -85,B 0,C 180,E1 -14127.624,E2 -14127.624} C_VEL
LIN {X 0,Y 339.007,Z 477.288,A -85,B 0,C 180,E1 -14128.812,E2 -14128.812} C_VEL
LIN {X 0,Y 339.007,Z 477.288,A -85,B 0,C 180,E1 -14131.188,E2 -14131.188} C_VEL
LIN {X 0,Y 338.999,Z 476.699,A -85,B 0,C 180,E1 -14132.376,E2 -14132.376} C_VEL
LIN {X 0,Y 339.064,Z 474.252,A -85,B 0,C 180,E1 -14134.756,E2 -14134.756} C_VEL
LIN {X 0,Y 339.17,Z 471.302,A -85,B 0,C 180,E1 -14136.544,E2 -14136.544} C_VEL
LIN {X 0,Y 339.512,Z 467.314,A -85,B 0,C 180,E1 -14138.332,E2 -14138.332} C_VEL
LIN {X 0,Y 339.996,Z 462.183,A -85,B 0,C 180,E1 -14140.119,E2 -14140.119} C_VEL
LIN {X 0,Y 340.566,Z 456.92,A -85,B 0,C 180,E1 -14141.607,E2 -14141.607} C_VEL
LIN {X 0,Y 341.387,Z 450.603,A -85,B 0,C 180,E1 -14143.088,E2 -14143.088} C_VEL
LIN {X 0,Y 342.124,Z 444.652,A -85,B 0,C 180,E1 -14144.271,E2 -14144.271} C_VEL
LIN {X 0,Y 343.139,Z 436.709,A -85,B 0,C 180,E1 -14145.603,E2 -14145.603} C_VEL
LIN {X 0,Y 343.984,Z 429.545,A -85,B 0,C 180,E1 -14146.621,E2 -14146.621} C_VEL
LIN {X 0,Y 345.017,Z 421.034,A -85,B 0,C 180,E1 -14147.638,E2 -14147.638} C_VEL
LIN {X 0,Y 345.991,Z 412.319,A -85,B 0,C 180,E1 -14148.505,E2 -14148.505} C_VEL
LIN {X 0,Y 346.916,Z 402.561,A -85,B 0,C 180,E1 -14149.297,E2 -14149.297} C_VEL
LIN {X 0,Y 347.715,Z 393.769,A -85,B 0,C 180,E1 -14149.865,E2 -14149.865} C_VEL
LIN {X 0,Y 348.442,Z 383.842,A -85,B 0,C 180,E1 -14150.361,E2 -14150.361} C_VEL
LIN {X 0,Y 348.952,Z 373.987,A -85,B 0,C 180,E1 -14150.715,E2 -14150.715} C_VEL
LIN {X 0,Y 349.494,Z 349.163,A -85,B 0,C 180,E1 -14151.264,E2 -14151.264} C_VEL
LIN {X 0,Y 350.144,Z 303.53,A -85,B 0,C 180,E1 -14152.208,E2 -14152.208} C_VEL
LIN {X 0,Y 345.638,Z 278.655,A -85,B 0,C 180,E1 -14153.059,E2 -14153.059} C_VEL
LIN {X 0,Y 343.087,Z 266.644,A -85,B 0,C 180,E1 -14153.545,E2 -14153.545} C_VEL
LIN {X 0,Y 343.301,Z 264.424,A -85,B 0,C 180,E1 -14154.169,E2 -14154.169} C_VEL
LIN {X 0,Y 344.091,Z 257.955,A -85,B 0,C 180,E1 -14156.267,E2 -14156.267} C_VEL
LIN {X 0,Y 343.273,Z 251.971,A -85,B 0,C 180,E1 -14158.313,E2 -14158.313} C_VEL
LIN {X 0,Y 341.393,Z 242.597,A -85,B 0,C 180,E1 -14161.622,E2 -14161.622} C_VEL
LIN {X 0,Y 340.731,Z 239.564,A -85,B 0,C 180,E1 -14162.781,E2 -14162.781} C_VEL
LIN {X 0,Y 340.712,Z 239.533,A -85,B 0,C 180,E1 -14166.44,E2 -14166.44} C_VEL
LIN {X 0,Y 340.7,Z 239.523,A -85,B 0,C 180,E1 -14169.752,E2 -14169.752} C_VEL
LIN {X 0,Y 340.678,Z 239.547,A -85,B 0,C 180,E1 -14172.904,E2 -14172.904} C_VEL
LIN {X 0,Y 340.677,Z 239.547,A -85,B 0,C 180,E1 -14177.095,E2 -14177.095} C_VEL
LIN {X 0,Y 340.7,Z 239.534,A -85,B 0,C 180,E1 -14180.247,E2 -14180.247} C_VEL
LIN {X 0,Y 340.709,Z 239.543,A -85,B 0,C 180,E1 -14183.559,E2 -14183.559} C_VEL
LIN {X 0,Y 340.693,Z 239.528,A -85,B 0,C 180,E1 -14186.153,E2 -14186.153} C_VEL
LIN {X 0,Y 340.742,Z 239.537,A -85,B 0,C 180,E1 -14190.329,E2 -14190.329} C_VEL
LIN {X 0,Y 340.804,Z 239.509,A -85,B 0,C 180,E1 -14193.019,E2 -14193.019} C_VEL
LIN {X 0,Y 340.755,Z 239.535,A -85,B 0,C 180,E1 -14195.638,E2 -14195.638} C_VEL
LIN {X 0,Y 340.746,Z 239.524,A -85,B 0,C 180,E1 -14199.473,E2 -14199.473} C_VEL
LIN {X 0,Y 340.792,Z 239.507,A -85,B 0,C 180,E1 -14201.98,E2 -14201.98} C_VEL
LIN {X 0,Y 340.87,Z 239.521,A -85,B 0,C 180,E1 -14205.704,E2 -14205.704} C_VEL
LIN {X 0,Y 340.848,Z 239.499,A -85,B 0,C 180,E1 -14209.305,E2 -14209.305} C_VEL
LIN {X 0,Y 341.016,Z 239.494,A -85,B 0,C 180,E1 -14212.896,E2 -14212.896} C_VEL
LIN {X 0,Y 341.167,Z 239.477,A -85,B 0,C 180,E1 -14217.638,E2 -14217.638} C_VEL
LIN {X 0,Y 341.275,Z 239.441,A -85,B 0,C 180,E1 -14219.999,E2 -14219.999} C_VEL
LIN {X 0,Y 341.168,Z 239.471,A -85,B 0,C 180,E1 -14222.361,E2 -14222.361} C_VEL
LIN {X 0,Y 341.057,Z 239.492,A -85,B 0,C 180,E1 -14227.101,E2 -14227.101} C_VEL
LIN {X 0,Y 340.87,Z 239.495,A -85,B 0,C 180,E1 -14230.693,E2 -14230.693} C_VEL
LIN {X 0,Y 340.861,Z 239.526,A -85,B 0,C 180,E1 -14234.324,E2 -14234.324} C_VEL
LIN {X 0,Y 340.835,Z 239.502,A -85,B 0,C 180,E1 -14238.466,E2 -14238.466} C_VEL
LIN {X 0,Y 340.715,Z 239.537,A -85,B 0,C 180,E1 -14241.841,E2 -14241.841} C_VEL
LIN {X 0,Y 340.769,Z 239.528,A -85,B 0,C 180,E1 -14245.664,E2 -14245.664} C_VEL
LIN {X 0,Y 340.738,Z 239.521,A -85,B 0,C 180,E1 -14248.319,E2 -14248.319} C_VEL
LIN {X 0,Y 340.701,Z 239.545,A -85,B 0,C 180,E1 -14251.044,E2 -14251.044} C_VEL
LIN {X 0,Y 340.715,Z 239.53,A -85,B 0,C 180,E1 -14255.278,E2 -14255.278} C_VEL
LIN {X 0,Y 340.709,Z 239.544,A -85,B 0,C 180,E1 -14258.386,E2 -14258.386} C_VEL
LIN {X 0,Y 340.723,Z 239.53,A -85,B 0,C 180,E1 -14261.303,E2 -14261.303} C_VEL
LIN {X 0,Y 340.74,Z 239.535,A -85,B 0,C 180,E1 -14264.528,E2 -14264.528} C_VEL
LIN {X 0,Y 340.695,Z 239.505,A -85,B 0,C 180,E1 -14268.692,E2 -14268.692} C_VEL
LIN {X 0,Y 340.735,Z 239.544,A -85,B 0,C 180,E1 -14271.773,E2 -14271.773} C_VEL
LIN {X 0,Y 340.719,Z 239.515,A -85,B 0,C 180,E1 -14275.595,E2 -14275.595} C_VEL
LIN {X 0,Y 340.694,Z 239.544,A -85,B 0,C 180,E1 -14278.955,E2 -14278.955} C_VEL
LIN {X 0,Y 340.773,Z 239.536,A -85,B 0,C 180,E1 -14282.475,E2 -14282.475} C_VEL
LIN {X 0,Y 340.752,Z 239.541,A -85,B 0,C 180,E1 -14285.638,E2 -14285.638} C_VEL
LIN {X 0,Y 340.749,Z 239.652,A -85,B 0,C 180,E1 -14287.813,E2 -14287.813} C_VEL
LIN {X 0,Y 340.931,Z 240.489,A -85,B 0,C 180,E1 -14288.111,E2 -14288.111} C_VEL
LIN {X 0,Y 342.359,Z 243.226,A -85,B 0,C 180,E1 -14288.51,E2 -14288.51} C_VEL
LIN {X 0,Y 344.493,Z 245.251,A -85,B 0,C 180,E1 -14288.96,E2 -14288.96} C_VEL
LIN {X 0,Y 346.593,Z 248.461,A -85,B 0,C 180,E1 -14289.486,E2 -14289.486} C_VEL
LIN {X 0,Y 348.969,Z 250.836,A -85,B 0,C 180,E1 -14290.042,E2 -14290.042} C_VEL
LIN {X 0,Y 351.593,Z 254.186,A -85,B 0,C 180,E1 -14290.687,E2 -14290.687} C_VEL
LIN {X 0,Y 353.9,Z 256.464,A -85,B 0,C 180,E1 -14291.279,E2 -14291.279} C_VEL
LIN {X 0,Y 357.171,Z 260.314,A -85,B 0,C 180,E1 -14292.137,E2 -14292.137} C_VEL
LIN {X 0,Y 359.47,Z 262.422,A -85,B 0,C 180,E1 -14292.775,E2 -14292.775} C_VEL
LIN {X 0,Y 362.8,Z 266.101,A -85,B 0,C 180,E1 -14293.735,E2 -14293.735} C_VEL
LIN {X 0,Y 365.929,Z 268.726,A -85,B 0,C 180,E1 -14294.673,E2 -14294.673} C_VEL
LIN {X 0,Y 369.293,Z 272.447,A -85,B 0,C 180,E1 -14295.807,E2 -14295.807} C_VEL
LIN {X 0,Y 372.814,Z 275.224,A -85,B 0,C 180,E1 -14297.04,E2 -14297.04} C_VEL
LIN {X 0,Y 376.097,Z 278.712,A -85,B 0,C 180,E1 -14298.351,E2 -14298.351} C_VEL
LIN {X 0,Y 379.225,Z 281.011,A -85,B 0,C 180,E1 -14299.703,E2 -14299.703} C_VEL
LIN {X 0,Y 381.144,Z 282.14,A -85,B 0,C 180,E1 -14300.617,E2 -14300.617} C_VEL
LIN {X 0,Y 383.823,Z 285.321,A -85,B 0,C 180,E1 -14302.189,E2 -14302.189} C_VEL
LIN {X 0,Y 386.499,Z 287.403,A -85,B 0,C 180,E1 -14304.061,E2 -14304.061} C_VEL
LIN {X 0,Y 388.386,Z 288.412,A -85,B 0,C 180,E1 -14305.849,E2 -14305.849} C_VEL
LIN {X 0,Y 389.529,Z 288.797,A -85,B 0,C 180,E1 -14307.434,E2 -14307.434} C_VEL
LIN {X 0,Y 390.1,Z 289.221,A -85,B 0,C 180,E1 -14308.968,E2 -14308.968} C_VEL
LIN {X 0,Y 390.27,Z 289.151,A -85,B 0,C 180,E1 -14310,E2 -14310} C_VEL
